// TIA Portal V16 export
// export: Created 2021-11-12T13:32:19.7443046Z, ExportSetting WithDefaults, DisplayName Totally Integrated Automation Portal, DisplayVersion V16 Update 3, DisplayName TIA Portal Version Control Interface, DisplayVersion V16 Update 2, DisplayName TIA Portal Openness, DisplayVersion V16 Update 3, DisplayName SINAMICS Startdrive Advanced, DisplayVersion V16 Update 5, DisplayName SINAMICS Startdrive G130, G150, S120, S150, SINAMICS MV, S210, DisplayVersion V16 Update 5, DisplayName SINAMICS Startdrive G110M, G120, G120C, G120D, G120P, G115D, DisplayVersion V16 Update 5, DisplayName STEP 7 Professional, DisplayVersion V16 Update 3, DisplayName STEP 7 Safety, DisplayVersion V16, DisplayName WinCC UA Professional, DisplayVersion V16 Update 3
FUNCTION_BLOCK "Station1R5"   // FB33, LAD
{ S7_Optimized_Access := 'TRUE' }
VERSION : 0.1
// stored: AutoNumber true, IsIECCheckEnabled false, IsRetainMemResEnabled false, MemoryReserve 100, SetENOAutomatically false, UDAEnableTagReadback false
   VAR
      SF_RO01_Timeout : "STD_DI_Mon";   // Move timeout
      "SF_CL01-BG01_Alarm" { S7_SetPoint := 'True'} : "STD_DI_Mon";
      "SF_CL01-BG02_Alarm" { S7_SetPoint := 'True'} : "STD_DI_Mon";
      SF_RC01 : "STD_DriveRobotABB";
      SF_RO01 : "STD_RobotABB";
      SF_RobotGripper : "STD_RobotGripper";
      SS_Edge { ExternalAccessible := 'False'; ExternalVisible := 'False'; ExternalWritable := 'False'} : Array[0..100] of Bool;
   END_VAR
   VAR RETAIN
      SDIPartID : DInt;
      SI_PartType { S7_SetPoint := 'True'} : Int;
   END_VAR
   VAR
      SI_150RowNr : Int;   // Row number in map of station 150
      SI_150LineNr : Int;   // Line number in map of station 150
      SI_170RowNr : Int;   // Row number in map of station 170
      SI_170LineNr : Int;   // Line number in map of station 170
      SI_BSN1BeltExt : Int;   // BSN1 belt extension
      SB1PosFound150 : Bool;   // Take position in map of station 150 found
      SB1PosFound170 : Bool;   // Take position in map of station 170 found
      SB1ReqToChangeTool : Bool;   // Request from zone command to change tools
      SB1ChangeToolDone : Bool;   // Changing tool process done
      SB1CycleAutostop : Bool;   // Cycle autostop command
      SB1ServicePosReq { ExternalAccessible := 'False'; ExternalVisible := 'False'; ExternalWritable := 'False'} : Bool;   // Request to go to/from service position
      SB1RobotInitialized : Bool;   // Robot is initialized
   END_VAR
   VAR_TEMP
      TS_RC01 : "UDT_DriveRobotABBControl";   // Robot controller RC01 control
      TS_RO01 : "UDT_RobotABBControl";   // Robot RO01 control
      TI_BSNJobNr : UInt;
      TI_RowNr : Int;   // Transfer mat card according to row number
      TI_LineNr : Int;   // Transfer mat card according to line number
      TB1PwrOK : Bool;   // Power for this station is OK
      TB1HomePosReq : Bool;   // Request to go to home position
      TB1CtrlRun : Bool;   // Robot controller is running in automat
      TB1GripperFree : Bool;   // Gripper free - info from robot and data tracking
      TB1Take150 : Bool;   // Take parts from 150
      TB1Take170 : Bool;   // Take parts from 170
      TB1PutBSN : Bool;   // Put parts BSN
      TB1ChangeToolUpDown : Bool;   // Change tool from CL01 to CL02
      TB1ChangeToolDownUp : Bool;   // Change tool from CL02 to CL01
      TB1FreePosBSN : Bool;   // Free position in furnace was found
      TB1JobNr150 : Bool;
      TB1JobNr170 : Bool;
   END_VAR
   VAR CONSTANT
      CI_JobHome : UInt := 1;
      CI_JobService : UInt := 2;
      CI_ChangeToolUpDown : UInt := 11;
      CI_ChangeToolDownUp : UInt := 12;
      CI_JobTake150Pos1 : UInt := 101;
      CI_JobTake150Pos2 : UInt := 102;
      CI_JobTake150Pos3 : UInt := 103;
      CI_JobTake150Pos4 : UInt := 104;
      CI_JobTake150Pos5 : UInt := 105;
      CI_JobTake150Pos6 : UInt := 106;
      CI_JobTake150Pos7 : UInt := 107;
      CI_JobTake150Pos8 : UInt := 108;
      CI_JobTake150Pos9 : UInt := 109;
      CI_JobTake150Pos10 : UInt := 110;
      CI_JobTake150Pos11 : UInt := 111;
      CI_JobTake150Pos12 : UInt := 112;
      CI_JobTake170Pos1 : UInt := 201;
      CI_JobTake170Pos2 : UInt := 202;
      CI_JobTake170Pos3 : UInt := 203;
      CI_JobTake170Pos4 : UInt := 204;
      CI_JobTake170Pos5 : UInt := 205;
      CI_JobTake170Pos6 : UInt := 206;
      CI_JobTake170Pos7 : UInt := 207;
      CI_JobTake170Pos8 : UInt := 208;
      CI_JobTake170Pos9 : UInt := 209;
      CI_JobTake170Pos10 : UInt := 210;
      CI_JobTake170Pos11 : UInt := 211;
      CI_JobTake170Pos12 : UInt := 212;
      CI_JobPutR12L12 : UInt := 301;
      CI_JobPutR12L23 : UInt := 302;
      CI_JobPutR12L34 : UInt := 303;
      CI_JobPutR12L45 : UInt := 304;
      CI_JobPutR23L12 : UInt := 305;
      CI_JobPutR23L23 : UInt := 306;
      CI_JobPutR23L34 : UInt := 307;
      CI_JobPutR23L45 : UInt := 308;
      CI_JobPutR34L12 : UInt := 309;
      CI_JobPutR34L23 : UInt := 310;
      CI_JobPutR34L34 : UInt := 311;
      CI_JobPutR34L45 : UInt := 312;
      CI_JobPutPosX : UInt := 313;
   END_VAR
   VAR_TEMP   // added for the SCL form of the ladder/FBD networks
      _w1 : Bool;
      _w2 : Bool;
      _w3 : Bool;
      _w4 : Bool;
      _w5 : Bool;
      _w6 : Bool;
      _w7 : Bool;
      _w8 : Bool;
      _w9 : Bool;
      _w10 : Bool;
      _w11 : Bool;
      _w12 : Bool;
      _w13 : Bool;
      _w14 : Bool;
   END_VAR
BEGIN

REGION Network 1: Clear temporary variables
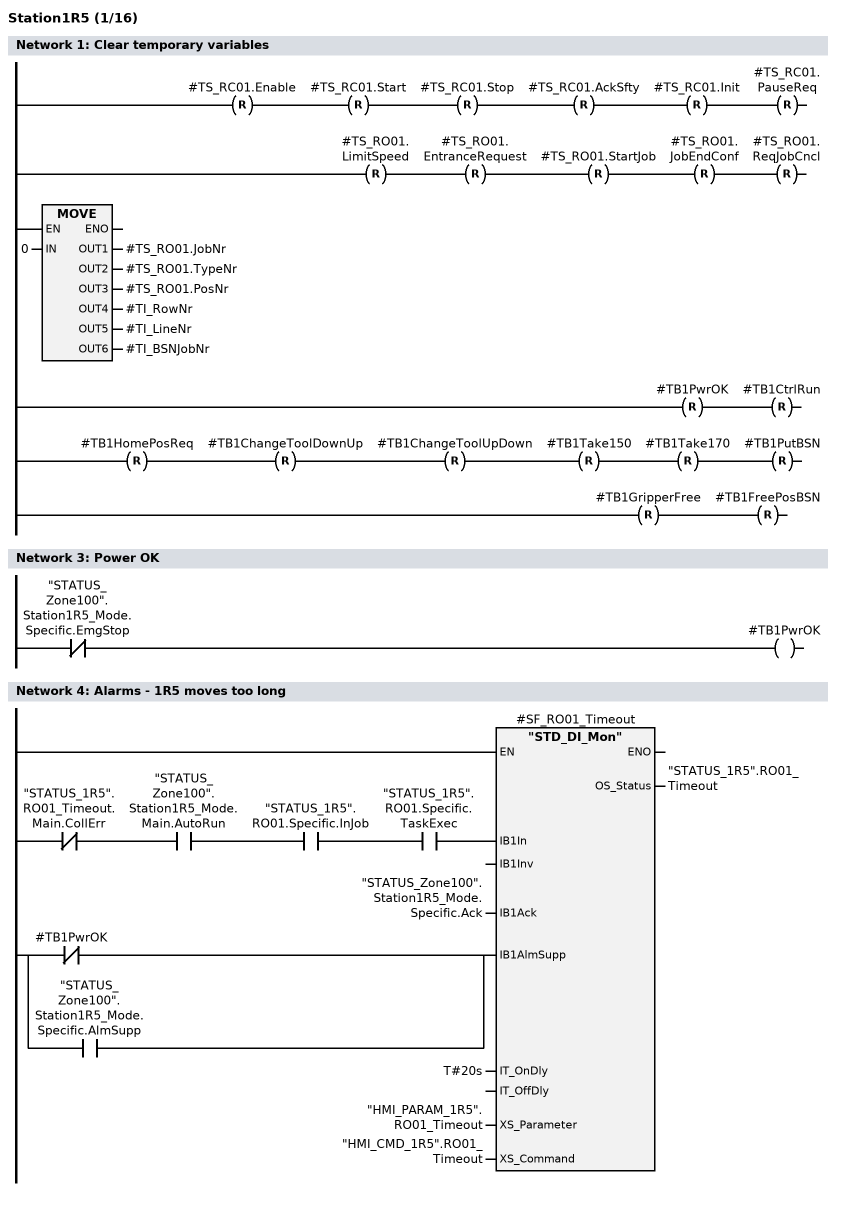
   RUNG wire#powerrail
      R_Coil( #TS_RC01.Enable )
      R_Coil( #TS_RC01.Start )
      R_Coil( #TS_RC01.Stop )
      R_Coil( #TS_RC01.AckSfty )
      R_Coil( #TS_RC01.Init )
      R_Coil( #TS_RC01.PauseReq )
   END_RUNG
   RUNG wire#powerrail
      R_Coil( #TS_RO01.LimitSpeed )
      R_Coil( #TS_RO01.EntranceRequest )
      R_Coil( #TS_RO01.StartJob )
      R_Coil( #TS_RO01.JobEndConf )
      R_Coil( #TS_RO01.ReqJobCncl )
   END_RUNG
   RUNG wire#powerrail
      Move(in := 0, out1 => #TS_RO01.JobNr, out2 => #TS_RO01.TypeNr, out3 => #TS_RO01.PosNr, out4 => #TI_RowNr, out5 => #TI_LineNr, out6 => #TI_BSNJobNr)
   END_RUNG
   RUNG wire#powerrail
      R_Coil( #TB1PwrOK )
      R_Coil( #TB1CtrlRun )
   END_RUNG
   RUNG wire#powerrail
      R_Coil( #TB1HomePosReq )
      R_Coil( #TB1ChangeToolDownUp )
      R_Coil( #TB1ChangeToolUpDown )
      R_Coil( #TB1Take150 )
      R_Coil( #TB1Take170 )
      R_Coil( #TB1PutBSN )
   END_RUNG
   RUNG wire#powerrail
      R_Coil( #TB1GripperFree )
      R_Coil( #TB1FreePosBSN )
   END_RUNG
   // the same network as SCL:
   #TS_RC01.Enable := FALSE;
   #TS_RC01.Start := FALSE;
   #TS_RC01.Stop := FALSE;
   #TS_RC01.AckSfty := FALSE;
   #TS_RC01.Init := FALSE;
   #TS_RC01.PauseReq := FALSE;
   #TS_RO01.LimitSpeed := FALSE;
   #TS_RO01.EntranceRequest := FALSE;
   #TS_RO01.StartJob := FALSE;
   #TS_RO01.JobEndConf := FALSE;
   #TS_RO01.ReqJobCncl := FALSE;
   #TS_RO01.JobNr := 0;
   #TS_RO01.TypeNr := 0;
   #TS_RO01.PosNr := 0;
   #TI_RowNr := 0;
   #TI_LineNr := 0;
   #TI_BSNJobNr := 0;
   #TB1PwrOK := FALSE;
   #TB1CtrlRun := FALSE;
   #TB1HomePosReq := FALSE;
   #TB1ChangeToolDownUp := FALSE;
   #TB1ChangeToolUpDown := FALSE;
   #TB1Take150 := FALSE;
   #TB1Take170 := FALSE;
   #TB1PutBSN := FALSE;
   #TB1GripperFree := FALSE;
   #TB1FreePosBSN := FALSE;
END_REGION

REGION Network 2: *************** Alarms ***************
END_REGION

REGION Network 3: Power OK
   RUNG wire#powerrail
      I_Contact( "STATUS_Zone100".Station1R5_Mode.Specific.EmgStop )
      Coil( #TB1PwrOK )
   END_RUNG
   // the same network as SCL:
   #TB1PwrOK := NOT "STATUS_Zone100".Station1R5_Mode.Specific.EmgStop;
END_REGION

REGION Network 4: Alarms - 1R5 moves too long
   RUNG wire#powerrail
      #SF_RO01_Timeout(IB1In := wire#w1, IB1AlmSupp := wire#w2, IB1Inv :=, IB1Ack := "STATUS_Zone100".Station1R5_Mode.Specific.Ack, IT_OnDly := T#20s, IT_OffDly :=, XS_Parameter := "HMI_PARAM_1R5".RO01_Timeout, XS_Command := "HMI_CMD_1R5".RO01_Timeout, OS_Status => "STATUS_1R5".RO01_Timeout)
   END_RUNG
   RUNG wire#powerrail
      I_Contact( "STATUS_1R5".RO01_Timeout.Main.CollErr )
      Contact( "STATUS_Zone100".Station1R5_Mode.Main.AutoRun )
      Contact( "STATUS_1R5".RO01.Specific.InJob )
      Contact( "STATUS_1R5".RO01.Specific.TaskExec )
   END_RUNG wire#w1
   RUNG wire#powerrail
      I_Contact( #TB1PwrOK )
   END_RUNG wire#w2
   RUNG wire#powerrail
      Contact( "STATUS_Zone100".Station1R5_Mode.Specific.AlmSupp )
   END_RUNG wire#w2
   // the same network as SCL:
   #SF_RO01_Timeout(IB1In := NOT "STATUS_1R5".RO01_Timeout.Main.CollErr AND "STATUS_Zone100".Station1R5_Mode.Main.AutoRun AND "STATUS_1R5".RO01.Specific.InJob AND "STATUS_1R5".RO01.Specific.TaskExec,   // "STD_DI_Mon"
                    IB1Ack := "STATUS_Zone100".Station1R5_Mode.Specific.Ack,
                    IB1AlmSupp := NOT #TB1PwrOK OR "STATUS_Zone100".Station1R5_Mode.Specific.AlmSupp,
                    IT_OnDly := T#20s,
                    XS_Parameter := "HMI_PARAM_1R5".RO01_Timeout,
                    XS_Command := "HMI_CMD_1R5".RO01_Timeout,
                    OS_Status => "STATUS_1R5".RO01_Timeout);
END_REGION

REGION Network 5: Sensor alarms - CL01
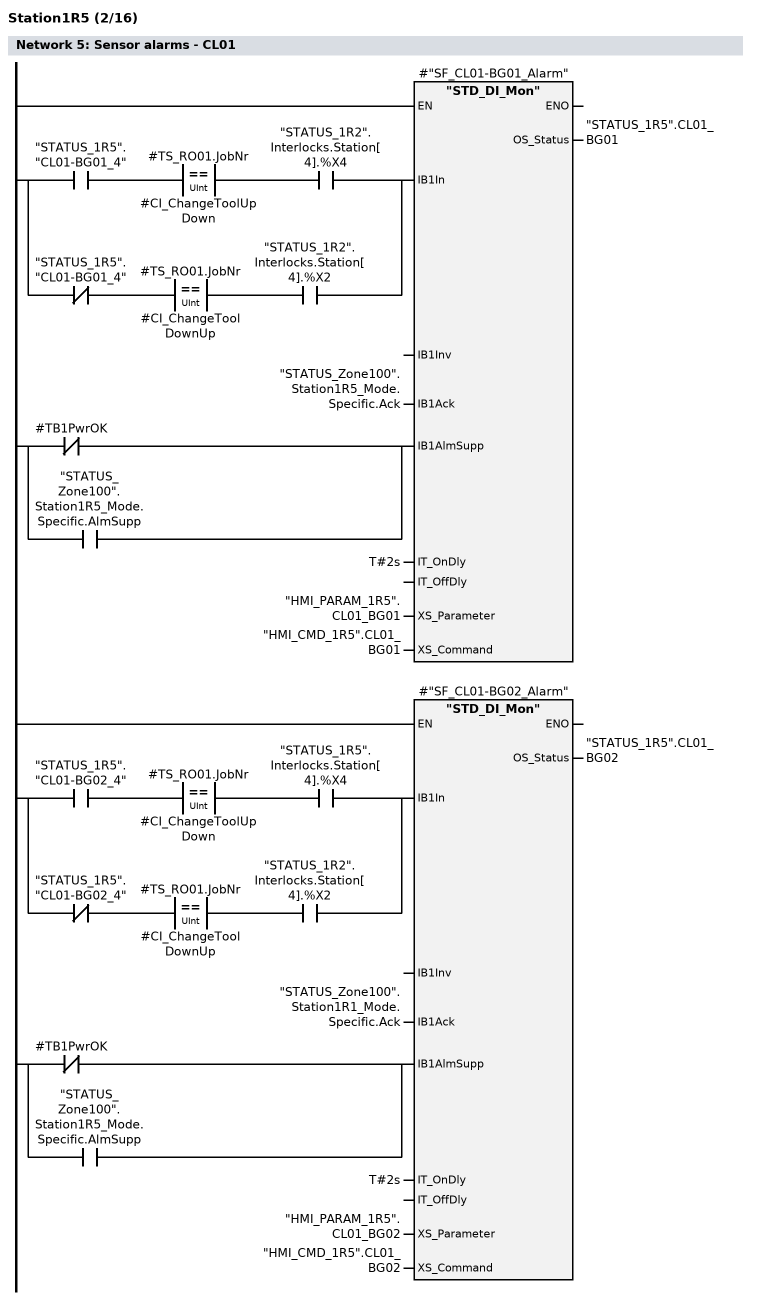
   RUNG wire#powerrail
      #"SF_CL01-BG01_Alarm"(IB1In := wire#w1, IB1AlmSupp := wire#w2, IB1Inv :=, IB1Ack := "STATUS_Zone100".Station1R5_Mode.Specific.Ack, IT_OnDly := T#2s, IT_OffDly :=, XS_Parameter := "HMI_PARAM_1R5".CL01_BG01, XS_Command := "HMI_CMD_1R5".CL01_BG01, OS_Status => "STATUS_1R5".CL01_BG01)
   END_RUNG
   RUNG wire#powerrail
      Contact( "STATUS_1R5"."CL01-BG01_4" )
      { S7_Templates := "SrcType := UInt" } EQ_Contact(in1 := #TS_RO01.JobNr, in2 := #CI_ChangeToolUpDown)
      Contact( "STATUS_1R2".Interlocks.Station[4].%X4 )
   END_RUNG wire#w1
   RUNG wire#powerrail
      I_Contact( "STATUS_1R5"."CL01-BG01_4" )
      { S7_Templates := "SrcType := UInt" } EQ_Contact(in1 := #TS_RO01.JobNr, in2 := #CI_ChangeToolDownUp)
      Contact( "STATUS_1R2".Interlocks.Station[4].%X2 )
   END_RUNG wire#w1
   RUNG wire#powerrail
      I_Contact( #TB1PwrOK )
   END_RUNG wire#w2
   RUNG wire#powerrail
      Contact( "STATUS_Zone100".Station1R5_Mode.Specific.AlmSupp )
   END_RUNG wire#w2
   RUNG wire#powerrail
      #"SF_CL01-BG02_Alarm"(IB1In := wire#w3, IB1AlmSupp := wire#w4, IB1Inv :=, IB1Ack := "STATUS_Zone100".Station1R1_Mode.Specific.Ack, IT_OnDly := T#2s, IT_OffDly :=, XS_Parameter := "HMI_PARAM_1R5".CL01_BG02, XS_Command := "HMI_CMD_1R5".CL01_BG02, OS_Status => "STATUS_1R5".CL01_BG02)
   END_RUNG
   RUNG wire#powerrail
      Contact( "STATUS_1R5"."CL01-BG02_4" )
      { S7_Templates := "SrcType := UInt" } EQ_Contact(in1 := #TS_RO01.JobNr, in2 := #CI_ChangeToolUpDown)
      Contact( "STATUS_1R5".Interlocks.Station[4].%X4 )
   END_RUNG wire#w3
   RUNG wire#powerrail
      I_Contact( "STATUS_1R5"."CL01-BG02_4" )
      { S7_Templates := "SrcType := UInt" } EQ_Contact(in1 := #TS_RO01.JobNr, in2 := #CI_ChangeToolDownUp)
      Contact( "STATUS_1R2".Interlocks.Station[4].%X2 )
   END_RUNG wire#w3
   RUNG wire#powerrail
      I_Contact( #TB1PwrOK )
   END_RUNG wire#w4
   RUNG wire#powerrail
      Contact( "STATUS_Zone100".Station1R5_Mode.Specific.AlmSupp )
   END_RUNG wire#w4
   // the same network as SCL:
   #"SF_CL01-BG01_Alarm"(IB1In := ("STATUS_1R5"."CL01-BG01_4" AND (#TS_RO01.JobNr = #CI_ChangeToolUpDown) AND "STATUS_1R2".Interlocks.Station[4].%X4) OR (NOT "STATUS_1R5"."CL01-BG01_4" AND (#TS_RO01.JobNr = #CI_ChangeToolDownUp) AND "STATUS_1R2".Interlocks.Station[4].%X2),   // "STD_DI_Mon"
                         IB1Ack := "STATUS_Zone100".Station1R5_Mode.Specific.Ack,
                         IB1AlmSupp := NOT #TB1PwrOK OR "STATUS_Zone100".Station1R5_Mode.Specific.AlmSupp,
                         IT_OnDly := T#2s,
                         XS_Parameter := "HMI_PARAM_1R5".CL01_BG01,
                         XS_Command := "HMI_CMD_1R5".CL01_BG01,
                         OS_Status => "STATUS_1R5".CL01_BG01);
   #"SF_CL01-BG02_Alarm"(IB1In := ("STATUS_1R5"."CL01-BG02_4" AND (#TS_RO01.JobNr = #CI_ChangeToolUpDown) AND "STATUS_1R5".Interlocks.Station[4].%X4) OR (NOT "STATUS_1R5"."CL01-BG02_4" AND (#TS_RO01.JobNr = #CI_ChangeToolDownUp) AND "STATUS_1R2".Interlocks.Station[4].%X2),   // "STD_DI_Mon"
                         IB1Ack := "STATUS_Zone100".Station1R1_Mode.Specific.Ack,
                         IB1AlmSupp := NOT #TB1PwrOK OR "STATUS_Zone100".Station1R5_Mode.Specific.AlmSupp,
                         IT_OnDly := T#2s,
                         XS_Parameter := "HMI_PARAM_1R5".CL01_BG02,
                         XS_Command := "HMI_CMD_1R5".CL01_BG02,
                         OS_Status => "STATUS_1R5".CL01_BG02);
END_REGION

REGION Network 6: *************** Controller RC01 ***************
END_REGION

REGION Network 7: Controller RC01 - control
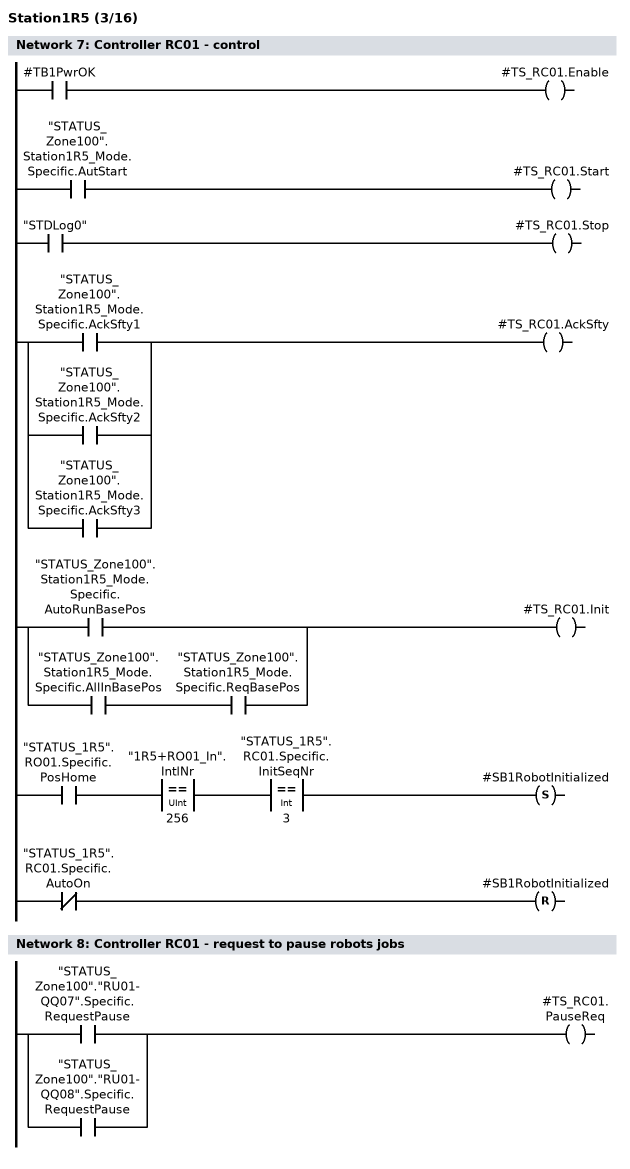
   RUNG wire#powerrail
      Contact( #TB1PwrOK )
      Coil( #TS_RC01.Enable )
   END_RUNG
   RUNG wire#powerrail
      Contact( "STATUS_Zone100".Station1R5_Mode.Specific.AutStart )
      Coil( #TS_RC01.Start )
   END_RUNG
   RUNG wire#powerrail
      Contact( "STDLog0" )
      Coil( #TS_RC01.Stop )
   END_RUNG
   RUNG wire#powerrail
      Contact( "STATUS_Zone100".Station1R5_Mode.Specific.AckSfty1 )
      wire#w1
      Coil( #TS_RC01.AckSfty )
   END_RUNG
   RUNG wire#powerrail
      Contact( "STATUS_Zone100".Station1R5_Mode.Specific.AckSfty2 )
   END_RUNG wire#w1
   RUNG wire#powerrail
      Contact( "STATUS_Zone100".Station1R5_Mode.Specific.AckSfty3 )
   END_RUNG wire#w1
   RUNG wire#powerrail
      Contact( "STATUS_Zone100".Station1R5_Mode.Specific.AutoRunBasePos )
      wire#w2
      Coil( #TS_RC01.Init )
   END_RUNG
   RUNG wire#powerrail
      Contact( "STATUS_Zone100".Station1R5_Mode.Specific.AllInBasePos )
      Contact( "STATUS_Zone100".Station1R5_Mode.Specific.ReqBasePos )
   END_RUNG wire#w2
   RUNG wire#powerrail
      Contact( "STATUS_1R5".RO01.Specific.PosHome )
      { S7_Templates := "SrcType := UInt" } EQ_Contact(in1 := "1R5+RO01_In".IntlNr, in2 := 256)
      { S7_Templates := "SrcType := Int" } EQ_Contact(in1 := "STATUS_1R5".RC01.Specific.InitSeqNr, in2 := 3)
      S_Coil( #SB1RobotInitialized )
   END_RUNG
   RUNG wire#powerrail
      I_Contact( "STATUS_1R5".RC01.Specific.AutoOn )
      R_Coil( #SB1RobotInitialized )
   END_RUNG
   // the same network as SCL:
   #TS_RC01.Enable := #TB1PwrOK;
   #TS_RC01.Start := "STATUS_Zone100".Station1R5_Mode.Specific.AutStart;
   #TS_RC01.Stop := "STDLog0";
   #TS_RC01.AckSfty := "STATUS_Zone100".Station1R5_Mode.Specific.AckSfty1 OR "STATUS_Zone100".Station1R5_Mode.Specific.AckSfty2 OR "STATUS_Zone100".Station1R5_Mode.Specific.AckSfty3;
   #TS_RC01.Init := "STATUS_Zone100".Station1R5_Mode.Specific.AutoRunBasePos OR ("STATUS_Zone100".Station1R5_Mode.Specific.AllInBasePos AND "STATUS_Zone100".Station1R5_Mode.Specific.ReqBasePos);
   IF "STATUS_1R5".RO01.Specific.PosHome AND ("1R5+RO01_In".IntlNr = 256) AND ("STATUS_1R5".RC01.Specific.InitSeqNr = 3) THEN
       #SB1RobotInitialized := TRUE;
   END_IF;
   IF NOT "STATUS_1R5".RC01.Specific.AutoOn THEN #SB1RobotInitialized := FALSE; END_IF;
END_REGION

REGION Network 8: Controller RC01 - request to pause robots jobs
   RUNG wire#powerrail
      Contact( "STATUS_Zone100"."RU01-QQ07".Specific.RequestPause )
      wire#w1
      Coil( #TS_RC01.PauseReq )
   END_RUNG
   RUNG wire#powerrail
      Contact( "STATUS_Zone100"."RU01-QQ08".Specific.RequestPause )
   END_RUNG wire#w1
   // the same network as SCL:
   #TS_RC01.PauseReq := "STATUS_Zone100"."RU01-QQ07".Specific.RequestPause OR "STATUS_Zone100"."RU01-QQ08".Specific.RequestPause;
END_REGION

REGION Network 9: Controller RC01 - main control
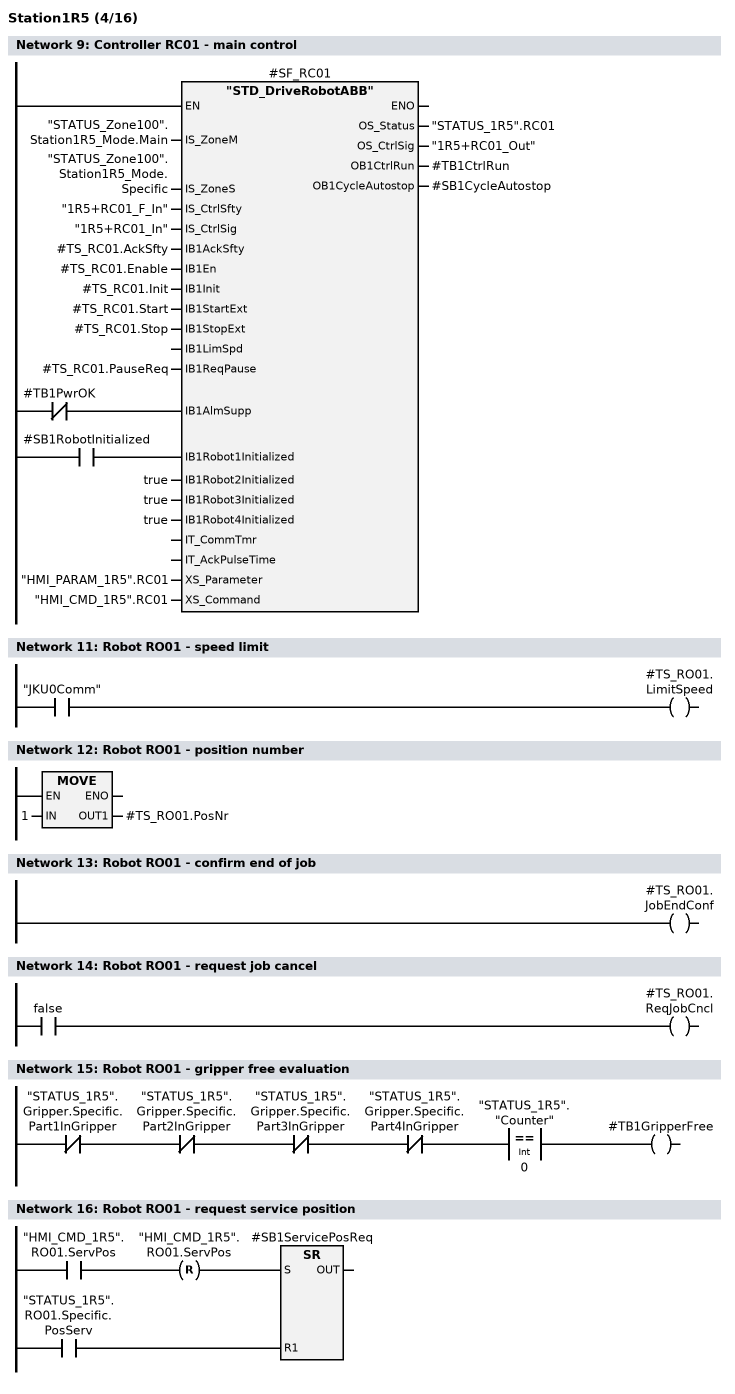
   RUNG wire#powerrail
      #SF_RC01(IB1AlmSupp := wire#w1, IB1Robot1Initialized := wire#w2, IS_ZoneM := "STATUS_Zone100".Station1R5_Mode.Main, IS_ZoneS := "STATUS_Zone100".Station1R5_Mode.Specific, IS_CtrlSfty := "1R5+RC01_F_In", IS_CtrlSig := "1R5+RC01_In", IB1AckSfty := #TS_RC01.AckSfty, IB1En := #TS_RC01.Enable, IB1Init := #TS_RC01.Init, IB1StartExt := #TS_RC01.Start, IB1StopExt := #TS_RC01.Stop, IB1LimSpd :=, IB1ReqPause := #TS_RC01.PauseReq, IB1Robot2Initialized := true, IB1Robot3Initialized := true, IB1Robot4Initialized := true, IT_CommTmr :=, IT_AckPulseTime :=, XS_Parameter := "HMI_PARAM_1R5".RC01, XS_Command := "HMI_CMD_1R5".RC01, OS_Status => "STATUS_1R5".RC01, OS_CtrlSig => "1R5+RC01_Out", OB1CtrlRun => #TB1CtrlRun, OB1CycleAutostop => #SB1CycleAutostop)
   END_RUNG
   RUNG wire#powerrail
      I_Contact( #TB1PwrOK )
   END_RUNG wire#w1
   RUNG wire#powerrail
      Contact( #SB1RobotInitialized )
   END_RUNG wire#w2
   // the same network as SCL:
   #SF_RC01(IS_ZoneM := "STATUS_Zone100".Station1R5_Mode.Main,   // "STD_DriveRobotABB"
            IS_ZoneS := "STATUS_Zone100".Station1R5_Mode.Specific,
            IS_CtrlSfty := "1R5+RC01_F_In",
            IS_CtrlSig := "1R5+RC01_In",
            IB1AckSfty := #TS_RC01.AckSfty,
            IB1En := #TS_RC01.Enable,
            IB1Init := #TS_RC01.Init,
            IB1StartExt := #TS_RC01.Start,
            IB1StopExt := #TS_RC01.Stop,
            IB1ReqPause := #TS_RC01.PauseReq,
            IB1AlmSupp := NOT #TB1PwrOK,
            IB1Robot1Initialized := #SB1RobotInitialized,
            IB1Robot2Initialized := true,
            IB1Robot3Initialized := true,
            IB1Robot4Initialized := true,
            XS_Parameter := "HMI_PARAM_1R5".RC01,
            XS_Command := "HMI_CMD_1R5".RC01,
            OS_Status => "STATUS_1R5".RC01,
            OS_CtrlSig => "1R5+RC01_Out",
            OB1CtrlRun => #TB1CtrlRun,
            OB1CycleAutostop => #SB1CycleAutostop);
END_REGION

REGION Network 10: *************** Robot RO01 ***************
END_REGION

REGION Network 11: Robot RO01 - speed limit
   RUNG wire#powerrail
      Contact( "JKU0Comm" )
      Coil( #TS_RO01.LimitSpeed )
   END_RUNG
   // the same network as SCL:
   #TS_RO01.LimitSpeed := "JKU0Comm";
END_REGION

REGION Network 12: Robot RO01 - position number
   RUNG wire#powerrail
      Move(in := 1, out1 => #TS_RO01.PosNr)
   END_RUNG
   // the same network as SCL:
   #TS_RO01.PosNr := 1;
END_REGION

REGION Network 13: Robot RO01 - confirm end of job
   RUNG wire#powerrail
      Coil( #TS_RO01.JobEndConf )
   END_RUNG
   // the same network as SCL:
   #TS_RO01.JobEndConf := TRUE;
END_REGION

REGION Network 14: Robot RO01 - request job cancel
   RUNG wire#powerrail
      Contact( false )
      Coil( #TS_RO01.ReqJobCncl )
   END_RUNG
   // the same network as SCL:
   #TS_RO01.ReqJobCncl := false;
END_REGION

REGION Network 15: Robot RO01 - gripper free evaluation
   RUNG wire#powerrail
      I_Contact( "STATUS_1R5".Gripper.Specific.Part1InGripper )
      I_Contact( "STATUS_1R5".Gripper.Specific.Part2InGripper )
      I_Contact( "STATUS_1R5".Gripper.Specific.Part3InGripper )
      I_Contact( "STATUS_1R5".Gripper.Specific.Part4InGripper )
      { S7_Templates := "SrcType := Int" } EQ_Contact(in1 := "STATUS_1R5"."Counter", in2 := 0)
      Coil( #TB1GripperFree )
   END_RUNG
   // the same network as SCL:
   #TB1GripperFree := NOT "STATUS_1R5".Gripper.Specific.Part1InGripper AND NOT "STATUS_1R5".Gripper.Specific.Part2InGripper AND NOT "STATUS_1R5".Gripper.Specific.Part3InGripper AND NOT "STATUS_1R5".Gripper.Specific.Part4InGripper AND ("STATUS_1R5"."Counter" = 0);
END_REGION

REGION Network 16: Robot RO01 - request service position
   RUNG wire#powerrail
      Contact( "HMI_CMD_1R5".RO01.ServPos )
      R_Coil( "HMI_CMD_1R5".RO01.ServPos )
      S_SR(operand := #SB1ServicePosReq, r1 := wire#w1)
   END_RUNG
   RUNG wire#powerrail
      Contact( "STATUS_1R5".RO01.Specific.PosServ )
   END_RUNG wire#w1
   // the same network as SCL:
   #_w1 := "HMI_CMD_1R5".RO01.ServPos;
   IF #_w1 THEN
       "HMI_CMD_1R5".RO01.ServPos := FALSE;
       #SB1ServicePosReq := TRUE;   // SR flip-flop
   END_IF;
   IF "STATUS_1R5".RO01.Specific.PosServ THEN #SB1ServicePosReq := FALSE; END_IF;
END_REGION

REGION Network 17: Robot RO01 - request home position
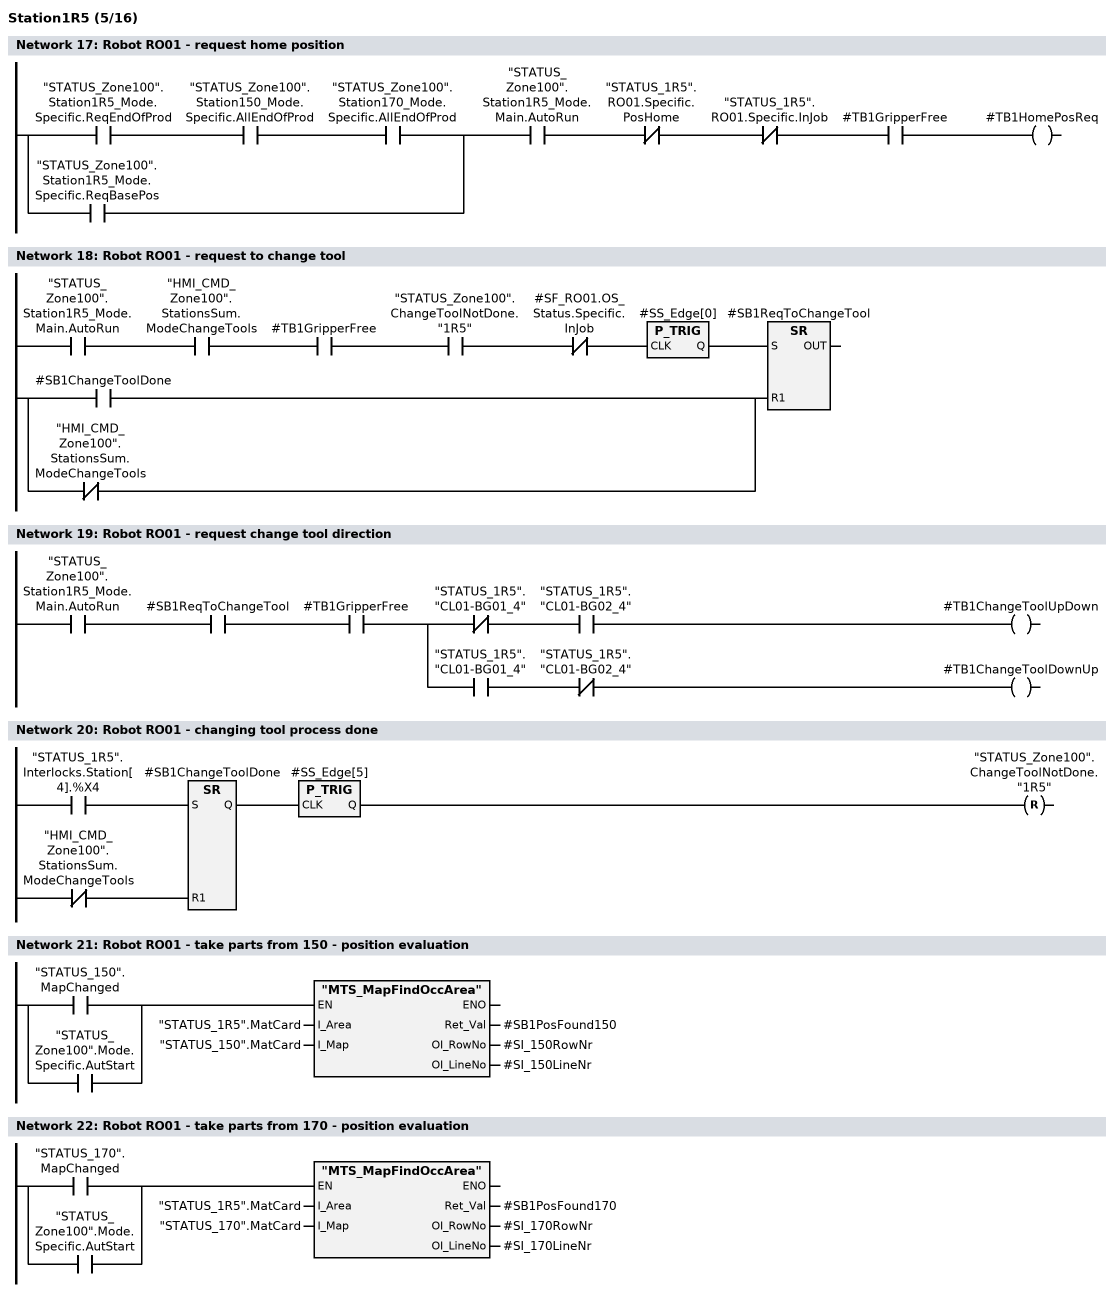
   RUNG wire#powerrail
      Contact( "STATUS_Zone100".Station1R5_Mode.Specific.ReqEndOfProd )
      Contact( "STATUS_Zone100".Station150_Mode.Specific.AllEndOfProd )
      Contact( "STATUS_Zone100".Station170_Mode.Specific.AllEndOfProd )
      wire#w1
      Contact( "STATUS_Zone100".Station1R5_Mode.Main.AutoRun )
      I_Contact( "STATUS_1R5".RO01.Specific.PosHome )
      I_Contact( "STATUS_1R5".RO01.Specific.InJob )
      Contact( #TB1GripperFree )
      Coil( #TB1HomePosReq )
   END_RUNG
   RUNG wire#powerrail
      Contact( "STATUS_Zone100".Station1R5_Mode.Specific.ReqBasePos )
   END_RUNG wire#w1
   // the same network as SCL:
   #TB1HomePosReq := (("STATUS_Zone100".Station1R5_Mode.Specific.ReqEndOfProd AND "STATUS_Zone100".Station150_Mode.Specific.AllEndOfProd AND "STATUS_Zone100".Station170_Mode.Specific.AllEndOfProd) OR "STATUS_Zone100".Station1R5_Mode.Specific.ReqBasePos) AND "STATUS_Zone100".Station1R5_Mode.Main.AutoRun AND NOT "STATUS_1R5".RO01.Specific.PosHome AND NOT "STATUS_1R5".RO01.Specific.InJob AND #TB1GripperFree;
END_REGION

REGION Network 18: Robot RO01 - request to change tool
   RUNG wire#powerrail
      Contact( "STATUS_Zone100".Station1R5_Mode.Main.AutoRun )
      Contact( "HMI_CMD_Zone100".StationsSum.ModeChangeTools )
      Contact( #TB1GripperFree )
      Contact( "STATUS_Zone100".ChangeToolNotDone."1R5" )
      I_Contact( #SF_RO01.OS_Status.Specific.InJob )
      P_Trig( #SS_Edge[0] )
      S_SR(operand := #SB1ReqToChangeTool, r1 := wire#w1)
   END_RUNG
   RUNG wire#powerrail
      Contact( #SB1ChangeToolDone )
   END_RUNG wire#w1
   RUNG wire#powerrail
      I_Contact( "HMI_CMD_Zone100".StationsSum.ModeChangeTools )
   END_RUNG wire#w1
   // the same network as SCL:
   #_w1 := "STATUS_Zone100".Station1R5_Mode.Main.AutoRun AND "HMI_CMD_Zone100".StationsSum.ModeChangeTools AND #TB1GripperFree AND "STATUS_Zone100".ChangeToolNotDone."1R5" AND NOT #SF_RO01.OS_Status.Specific.InJob;
   #_w2 := #_w1 AND NOT #SS_Edge[0];   // rising edge
   #SS_Edge[0] := #_w1;
   IF #_w2 THEN
       #SB1ReqToChangeTool := TRUE;   // SR flip-flop
   END_IF;
   IF #SB1ChangeToolDone OR NOT "HMI_CMD_Zone100".StationsSum.ModeChangeTools THEN
       #SB1ReqToChangeTool := FALSE;
   END_IF;
END_REGION

REGION Network 19: Robot RO01 - request change tool direction
   RUNG wire#powerrail
      Contact( "STATUS_Zone100".Station1R5_Mode.Main.AutoRun )
      Contact( #SB1ReqToChangeTool )
      Contact( #TB1GripperFree )
      wire#w1
      I_Contact( "STATUS_1R5"."CL01-BG01_4" )
      Contact( "STATUS_1R5"."CL01-BG02_4" )
      Coil( #TB1ChangeToolUpDown )
   END_RUNG
   RUNG wire#w1
      Contact( "STATUS_1R5"."CL01-BG01_4" )
      I_Contact( "STATUS_1R5"."CL01-BG02_4" )
      Coil( #TB1ChangeToolDownUp )
   END_RUNG
   // the same network as SCL:
   #_w1 := "STATUS_Zone100".Station1R5_Mode.Main.AutoRun AND #SB1ReqToChangeTool AND #TB1GripperFree;
   #TB1ChangeToolUpDown := #_w1 AND NOT "STATUS_1R5"."CL01-BG01_4" AND "STATUS_1R5"."CL01-BG02_4";
   #TB1ChangeToolDownUp := #_w1 AND "STATUS_1R5"."CL01-BG01_4" AND NOT "STATUS_1R5"."CL01-BG02_4";
END_REGION

REGION Network 20: Robot RO01 - changing tool process done
   RUNG wire#powerrail
      Contact( "STATUS_1R5".Interlocks.Station[4].%X4 )
      S_SR(operand := #SB1ChangeToolDone, r1 := wire#w1)
      P_Trig( #SS_Edge[5] )
      R_Coil( "STATUS_Zone100".ChangeToolNotDone."1R5" )
   END_RUNG
   RUNG wire#powerrail
      I_Contact( "HMI_CMD_Zone100".StationsSum.ModeChangeTools )
   END_RUNG wire#w1
   // the same network as SCL:
   IF "STATUS_1R5".Interlocks.Station[4].%X4 THEN
       #SB1ChangeToolDone := TRUE;   // SR flip-flop
   END_IF;
   IF NOT "HMI_CMD_Zone100".StationsSum.ModeChangeTools THEN #SB1ChangeToolDone := FALSE; END_IF;
   #_w1 := #SB1ChangeToolDone AND NOT #SS_Edge[5];   // rising edge
   #SS_Edge[5] := #SB1ChangeToolDone;
   IF #_w1 THEN "STATUS_Zone100".ChangeToolNotDone."1R5" := FALSE; END_IF;
END_REGION

REGION Network 21: Robot RO01 - take parts from 150 - position evaluation
   RUNG wire#powerrail
      Contact( "STATUS_150".MapChanged )
      wire#w1
      "MTS_MapFindOccArea"(I_Area := "STATUS_1R5".MatCard, I_Map := "STATUS_150".MatCard, Ret_Val => #SB1PosFound150, OI_RowNo => #SI_150RowNr, OI_LineNo => #SI_150LineNr)
   END_RUNG
   RUNG wire#powerrail
      Contact( "STATUS_Zone100".Mode.Specific.AutStart )
   END_RUNG wire#w1
   // the same network as SCL:
   IF "STATUS_150".MapChanged OR "STATUS_Zone100".Mode.Specific.AutStart THEN
       #SB1PosFound150 := "MTS_MapFindOccArea"(I_Area := "STATUS_1R5".MatCard,
                               I_Map := "STATUS_150".MatCard,
                               OI_RowNo => #SI_150RowNr,
                               OI_LineNo => #SI_150LineNr);
   END_IF;
END_REGION

REGION Network 22: Robot RO01 - take parts from 170 - position evaluation
   RUNG wire#powerrail
      Contact( "STATUS_170".MapChanged )
      wire#w1
      "MTS_MapFindOccArea"(I_Area := "STATUS_1R5".MatCard, I_Map := "STATUS_170".MatCard, Ret_Val => #SB1PosFound170, OI_RowNo => #SI_170RowNr, OI_LineNo => #SI_170LineNr)
   END_RUNG
   RUNG wire#powerrail
      Contact( "STATUS_Zone100".Mode.Specific.AutStart )
   END_RUNG wire#w1
   // the same network as SCL:
   IF "STATUS_170".MapChanged OR "STATUS_Zone100".Mode.Specific.AutStart THEN
       #SB1PosFound170 := "MTS_MapFindOccArea"(I_Area := "STATUS_1R5".MatCard,
                               I_Map := "STATUS_170".MatCard,
                               OI_RowNo => #SI_170RowNr,
                               OI_LineNo => #SI_170LineNr);
   END_IF;
END_REGION

REGION Network 23: Robot RO01 - table 150/170 - take command
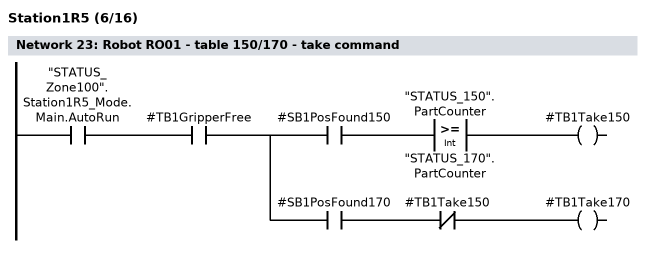
   RUNG wire#powerrail
      Contact( "STATUS_Zone100".Station1R5_Mode.Main.AutoRun )
      Contact( #TB1GripperFree )
      wire#w1
      Contact( #SB1PosFound150 )
      { S7_Templates := "SrcType := Int" } GE_Contact(in1 := "STATUS_150".PartCounter, in2 := "STATUS_170".PartCounter)
      Coil( #TB1Take150 )
   END_RUNG
   RUNG wire#w1
      Contact( #SB1PosFound170 )
      I_Contact( #TB1Take150 )
      Coil( #TB1Take170 )
   END_RUNG
   // the same network as SCL:
   #_w1 := "STATUS_Zone100".Station1R5_Mode.Main.AutoRun AND #TB1GripperFree;
   #TB1Take150 := #_w1 AND #SB1PosFound150 AND ("STATUS_150".PartCounter >= "STATUS_170".PartCounter);
   #TB1Take170 := #_w1 AND #SB1PosFound170 AND NOT #TB1Take150;
END_REGION

REGION Network 24: Robot RO01 - BSN1 position evaluation
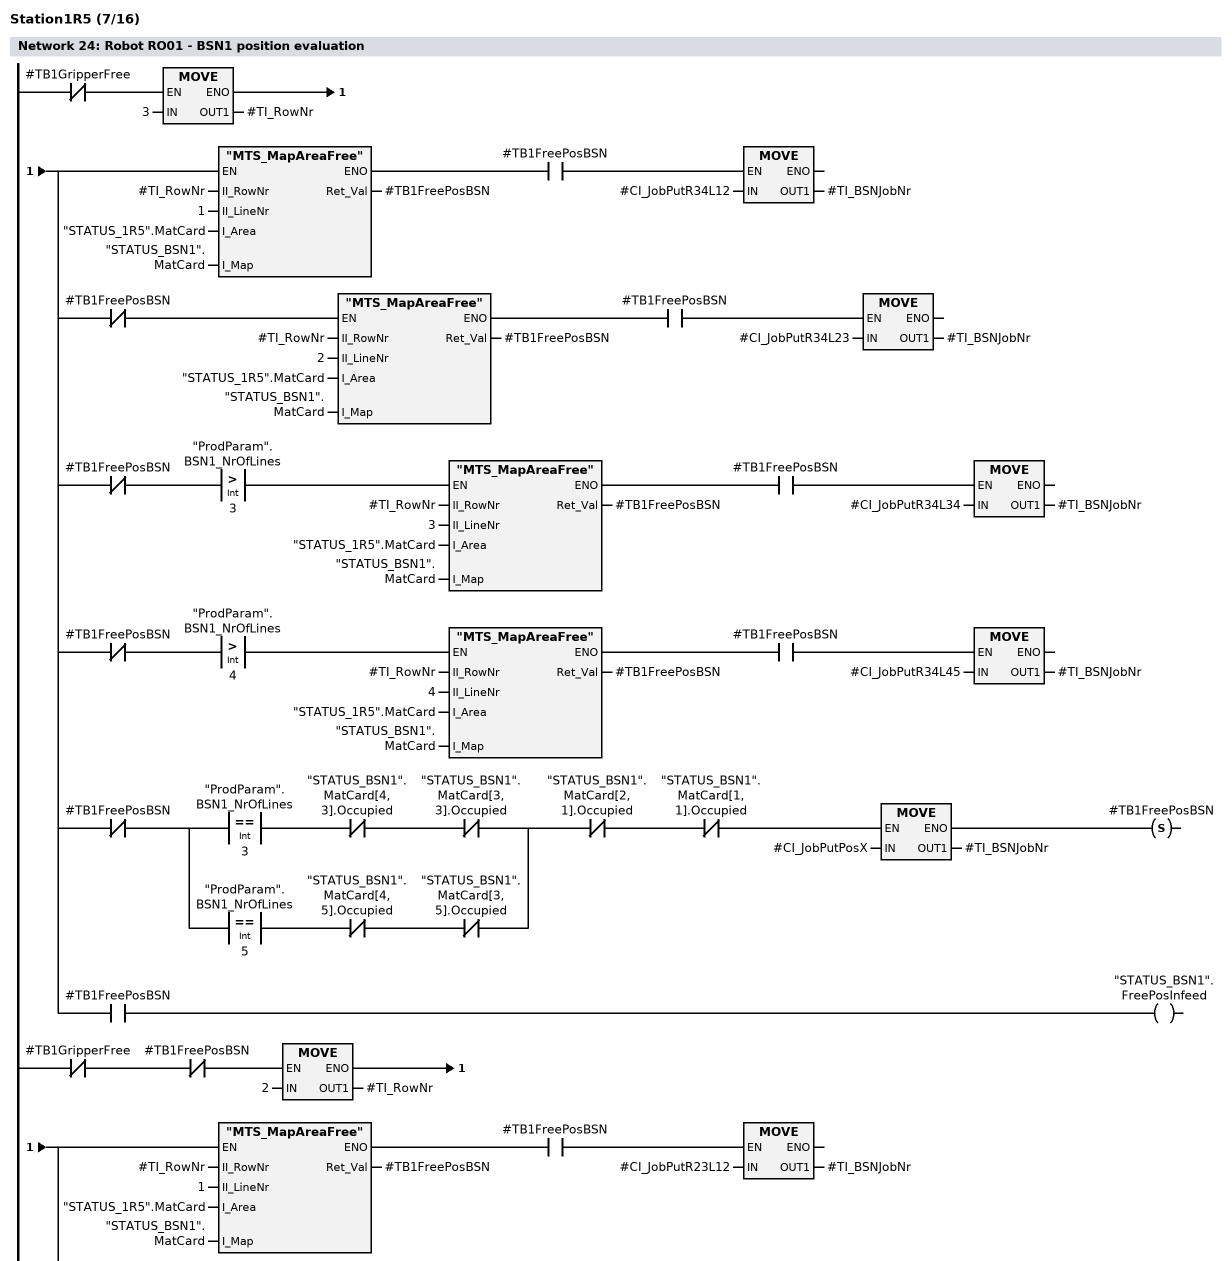
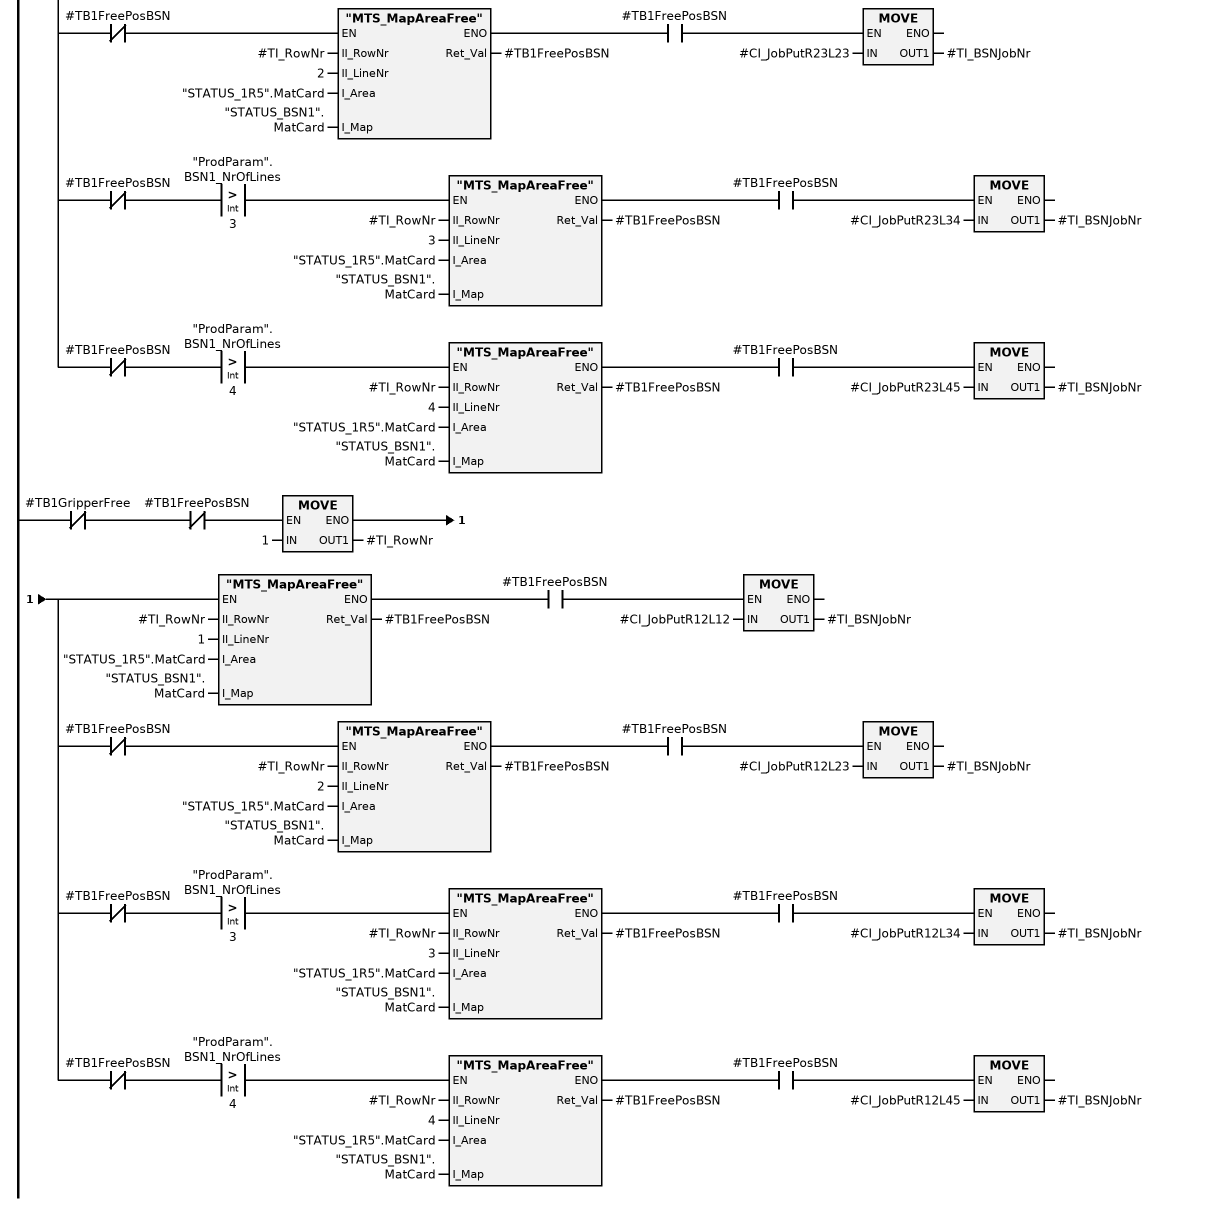
   RUNG wire#powerrail
      I_Contact( #TB1GripperFree )
      Move(in := 3, out1 => #TI_RowNr)
      wire#w1
      "MTS_MapAreaFree"(II_RowNr := #TI_RowNr, II_LineNr := 1, I_Area := "STATUS_1R5".MatCard, I_Map := "STATUS_BSN1".MatCard, Ret_Val => #TB1FreePosBSN)
      Contact( #TB1FreePosBSN )
      Move(in := #CI_JobPutR34L12, out1 => #TI_BSNJobNr)
   END_RUNG
   RUNG wire#w1
      I_Contact( #TB1FreePosBSN )
      "MTS_MapAreaFree"(II_RowNr := #TI_RowNr, II_LineNr := 2, I_Area := "STATUS_1R5".MatCard, I_Map := "STATUS_BSN1".MatCard, Ret_Val => #TB1FreePosBSN)
      Contact( #TB1FreePosBSN )
      Move(in := #CI_JobPutR34L23, out1 => #TI_BSNJobNr)
   END_RUNG
   RUNG wire#w1
      I_Contact( #TB1FreePosBSN )
      { S7_Templates := "SrcType := Int" } GT_Contact(in1 := "ProdParam".BSN1_NrOfLines, in2 := 3)
      "MTS_MapAreaFree"(II_RowNr := #TI_RowNr, II_LineNr := 3, I_Area := "STATUS_1R5".MatCard, I_Map := "STATUS_BSN1".MatCard, Ret_Val => #TB1FreePosBSN)
      Contact( #TB1FreePosBSN )
      Move(in := #CI_JobPutR34L34, out1 => #TI_BSNJobNr)
   END_RUNG
   RUNG wire#w1
      I_Contact( #TB1FreePosBSN )
      { S7_Templates := "SrcType := Int" } GT_Contact(in1 := "ProdParam".BSN1_NrOfLines, in2 := 4)
      "MTS_MapAreaFree"(II_RowNr := #TI_RowNr, II_LineNr := 4, I_Area := "STATUS_1R5".MatCard, I_Map := "STATUS_BSN1".MatCard, Ret_Val => #TB1FreePosBSN)
      Contact( #TB1FreePosBSN )
      Move(in := #CI_JobPutR34L45, out1 => #TI_BSNJobNr)
   END_RUNG
   RUNG wire#w1
      I_Contact( #TB1FreePosBSN )
      wire#w2
      { S7_Templates := "SrcType := Int" } EQ_Contact(in1 := "ProdParam".BSN1_NrOfLines, in2 := 3)
      I_Contact( "STATUS_BSN1".MatCard[4, 3].Occupied )
      I_Contact( "STATUS_BSN1".MatCard[3, 3].Occupied )
      wire#w3
      I_Contact( "STATUS_BSN1".MatCard[2, 1].Occupied )
      I_Contact( "STATUS_BSN1".MatCard[1, 1].Occupied )
      Move(in := #CI_JobPutPosX, out1 => #TI_BSNJobNr)
      S_Coil( #TB1FreePosBSN )
   END_RUNG
   RUNG wire#w2
      { S7_Templates := "SrcType := Int" } EQ_Contact(in1 := "ProdParam".BSN1_NrOfLines, in2 := 5)
      I_Contact( "STATUS_BSN1".MatCard[4, 5].Occupied )
      I_Contact( "STATUS_BSN1".MatCard[3, 5].Occupied )
   END_RUNG wire#w3
   RUNG wire#w1
      Contact( #TB1FreePosBSN )
      Coil( "STATUS_BSN1".FreePosInfeed )
   END_RUNG
   RUNG wire#powerrail
      I_Contact( #TB1GripperFree )
      I_Contact( #TB1FreePosBSN )
      Move(in := 2, out1 => #TI_RowNr)
      wire#w4
      "MTS_MapAreaFree"(II_RowNr := #TI_RowNr, II_LineNr := 1, I_Area := "STATUS_1R5".MatCard, I_Map := "STATUS_BSN1".MatCard, Ret_Val => #TB1FreePosBSN)
      Contact( #TB1FreePosBSN )
      Move(in := #CI_JobPutR23L12, out1 => #TI_BSNJobNr)
   END_RUNG
   RUNG wire#w4
      I_Contact( #TB1FreePosBSN )
      "MTS_MapAreaFree"(II_RowNr := #TI_RowNr, II_LineNr := 2, I_Area := "STATUS_1R5".MatCard, I_Map := "STATUS_BSN1".MatCard, Ret_Val => #TB1FreePosBSN)
      Contact( #TB1FreePosBSN )
      Move(in := #CI_JobPutR23L23, out1 => #TI_BSNJobNr)
   END_RUNG
   RUNG wire#w4
      I_Contact( #TB1FreePosBSN )
      { S7_Templates := "SrcType := Int" } GT_Contact(in1 := "ProdParam".BSN1_NrOfLines, in2 := 3)
      "MTS_MapAreaFree"(II_RowNr := #TI_RowNr, II_LineNr := 3, I_Area := "STATUS_1R5".MatCard, I_Map := "STATUS_BSN1".MatCard, Ret_Val => #TB1FreePosBSN)
      Contact( #TB1FreePosBSN )
      Move(in := #CI_JobPutR23L34, out1 => #TI_BSNJobNr)
   END_RUNG
   RUNG wire#w4
      I_Contact( #TB1FreePosBSN )
      { S7_Templates := "SrcType := Int" } GT_Contact(in1 := "ProdParam".BSN1_NrOfLines, in2 := 4)
      "MTS_MapAreaFree"(II_RowNr := #TI_RowNr, II_LineNr := 4, I_Area := "STATUS_1R5".MatCard, I_Map := "STATUS_BSN1".MatCard, Ret_Val => #TB1FreePosBSN)
      Contact( #TB1FreePosBSN )
      Move(in := #CI_JobPutR23L45, out1 => #TI_BSNJobNr)
   END_RUNG
   RUNG wire#powerrail
      I_Contact( #TB1GripperFree )
      I_Contact( #TB1FreePosBSN )
      Move(in := 1, out1 => #TI_RowNr)
      wire#w5
      "MTS_MapAreaFree"(II_RowNr := #TI_RowNr, II_LineNr := 1, I_Area := "STATUS_1R5".MatCard, I_Map := "STATUS_BSN1".MatCard, Ret_Val => #TB1FreePosBSN)
      Contact( #TB1FreePosBSN )
      Move(in := #CI_JobPutR12L12, out1 => #TI_BSNJobNr)
   END_RUNG
   RUNG wire#w5
      I_Contact( #TB1FreePosBSN )
      "MTS_MapAreaFree"(II_RowNr := #TI_RowNr, II_LineNr := 2, I_Area := "STATUS_1R5".MatCard, I_Map := "STATUS_BSN1".MatCard, Ret_Val => #TB1FreePosBSN)
      Contact( #TB1FreePosBSN )
      Move(in := #CI_JobPutR12L23, out1 => #TI_BSNJobNr)
   END_RUNG
   RUNG wire#w5
      I_Contact( #TB1FreePosBSN )
      { S7_Templates := "SrcType := Int" } GT_Contact(in1 := "ProdParam".BSN1_NrOfLines, in2 := 3)
      "MTS_MapAreaFree"(II_RowNr := #TI_RowNr, II_LineNr := 3, I_Area := "STATUS_1R5".MatCard, I_Map := "STATUS_BSN1".MatCard, Ret_Val => #TB1FreePosBSN)
      Contact( #TB1FreePosBSN )
      Move(in := #CI_JobPutR12L34, out1 => #TI_BSNJobNr)
   END_RUNG
   RUNG wire#w5
      I_Contact( #TB1FreePosBSN )
      { S7_Templates := "SrcType := Int" } GT_Contact(in1 := "ProdParam".BSN1_NrOfLines, in2 := 4)
      "MTS_MapAreaFree"(II_RowNr := #TI_RowNr, II_LineNr := 4, I_Area := "STATUS_1R5".MatCard, I_Map := "STATUS_BSN1".MatCard, Ret_Val => #TB1FreePosBSN)
      Contact( #TB1FreePosBSN )
      Move(in := #CI_JobPutR12L45, out1 => #TI_BSNJobNr)
   END_RUNG
   // the same network as SCL:
   IF NOT #TB1GripperFree THEN #TI_RowNr := 3; END_IF;
   #TB1FreePosBSN := "MTS_MapAreaFree"(EN := NOT #TB1GripperFree,
                           II_RowNr := #TI_RowNr,
                           II_LineNr := 1,
                           I_Area := "STATUS_1R5".MatCard,
                           I_Map := "STATUS_BSN1".MatCard,
                           ENO => #_w1);
   IF #_w1 AND #TB1FreePosBSN THEN #TI_BSNJobNr := #CI_JobPutR34L12; END_IF;
   #TB1FreePosBSN := "MTS_MapAreaFree"(EN := NOT #TB1GripperFree AND NOT #TB1FreePosBSN,
                           II_RowNr := #TI_RowNr,
                           II_LineNr := 2,
                           I_Area := "STATUS_1R5".MatCard,
                           I_Map := "STATUS_BSN1".MatCard,
                           ENO => #_w2);
   IF #_w2 AND #TB1FreePosBSN THEN #TI_BSNJobNr := #CI_JobPutR34L23; END_IF;
   #TB1FreePosBSN := "MTS_MapAreaFree"(EN := NOT #TB1GripperFree AND NOT #TB1FreePosBSN AND ("ProdParam".BSN1_NrOfLines > 3),
                           II_RowNr := #TI_RowNr,
                           II_LineNr := 3,
                           I_Area := "STATUS_1R5".MatCard,
                           I_Map := "STATUS_BSN1".MatCard,
                           ENO => #_w3);
   IF #_w3 AND #TB1FreePosBSN THEN #TI_BSNJobNr := #CI_JobPutR34L34; END_IF;
   #TB1FreePosBSN := "MTS_MapAreaFree"(EN := NOT #TB1GripperFree AND NOT #TB1FreePosBSN AND ("ProdParam".BSN1_NrOfLines > 4),
                           II_RowNr := #TI_RowNr,
                           II_LineNr := 4,
                           I_Area := "STATUS_1R5".MatCard,
                           I_Map := "STATUS_BSN1".MatCard,
                           ENO => #_w4);
   IF #_w4 AND #TB1FreePosBSN THEN #TI_BSNJobNr := #CI_JobPutR34L45; END_IF;
   IF NOT #TB1GripperFree AND NOT #TB1FreePosBSN AND ((("ProdParam".BSN1_NrOfLines = 3) AND NOT "STATUS_BSN1".MatCard[4, 3].Occupied AND NOT "STATUS_BSN1".MatCard[3, 3].Occupied) OR (("ProdParam".BSN1_NrOfLines = 5) AND NOT "STATUS_BSN1".MatCard[4, 5].Occupied AND NOT "STATUS_BSN1".MatCard[3, 5].Occupied)) AND NOT "STATUS_BSN1".MatCard[2, 1].Occupied AND NOT "STATUS_BSN1".MatCard[1, 1].Occupied THEN
       #TI_BSNJobNr := #CI_JobPutPosX;
       #TB1FreePosBSN := TRUE;
   END_IF;
   "STATUS_BSN1".FreePosInfeed := NOT #TB1GripperFree AND #TB1FreePosBSN;
   #_w5 := NOT #TB1GripperFree AND NOT #TB1FreePosBSN;
   IF #_w5 THEN #TI_RowNr := 2; END_IF;
   #TB1FreePosBSN := "MTS_MapAreaFree"(EN := #_w5,
                           II_RowNr := #TI_RowNr,
                           II_LineNr := 1,
                           I_Area := "STATUS_1R5".MatCard,
                           I_Map := "STATUS_BSN1".MatCard,
                           ENO => #_w6);
   IF #_w6 AND #TB1FreePosBSN THEN #TI_BSNJobNr := #CI_JobPutR23L12; END_IF;
   #TB1FreePosBSN := "MTS_MapAreaFree"(EN := #_w5 AND NOT #TB1FreePosBSN,
                           II_RowNr := #TI_RowNr,
                           II_LineNr := 2,
                           I_Area := "STATUS_1R5".MatCard,
                           I_Map := "STATUS_BSN1".MatCard,
                           ENO => #_w7);
   IF #_w7 AND #TB1FreePosBSN THEN #TI_BSNJobNr := #CI_JobPutR23L23; END_IF;
   #TB1FreePosBSN := "MTS_MapAreaFree"(EN := #_w5 AND NOT #TB1FreePosBSN AND ("ProdParam".BSN1_NrOfLines > 3),
                           II_RowNr := #TI_RowNr,
                           II_LineNr := 3,
                           I_Area := "STATUS_1R5".MatCard,
                           I_Map := "STATUS_BSN1".MatCard,
                           ENO => #_w8);
   IF #_w8 AND #TB1FreePosBSN THEN #TI_BSNJobNr := #CI_JobPutR23L34; END_IF;
   #TB1FreePosBSN := "MTS_MapAreaFree"(EN := #_w5 AND NOT #TB1FreePosBSN AND ("ProdParam".BSN1_NrOfLines > 4),
                           II_RowNr := #TI_RowNr,
                           II_LineNr := 4,
                           I_Area := "STATUS_1R5".MatCard,
                           I_Map := "STATUS_BSN1".MatCard,
                           ENO => #_w9);
   IF #_w9 AND #TB1FreePosBSN THEN #TI_BSNJobNr := #CI_JobPutR23L45; END_IF;
   #_w10 := NOT #TB1GripperFree AND NOT #TB1FreePosBSN;
   IF #_w10 THEN #TI_RowNr := 1; END_IF;
   #TB1FreePosBSN := "MTS_MapAreaFree"(EN := #_w10,
                           II_RowNr := #TI_RowNr,
                           II_LineNr := 1,
                           I_Area := "STATUS_1R5".MatCard,
                           I_Map := "STATUS_BSN1".MatCard,
                           ENO => #_w11);
   IF #_w11 AND #TB1FreePosBSN THEN #TI_BSNJobNr := #CI_JobPutR12L12; END_IF;
   #TB1FreePosBSN := "MTS_MapAreaFree"(EN := #_w10 AND NOT #TB1FreePosBSN,
                           II_RowNr := #TI_RowNr,
                           II_LineNr := 2,
                           I_Area := "STATUS_1R5".MatCard,
                           I_Map := "STATUS_BSN1".MatCard,
                           ENO => #_w12);
   IF #_w12 AND #TB1FreePosBSN THEN #TI_BSNJobNr := #CI_JobPutR12L23; END_IF;
   #TB1FreePosBSN := "MTS_MapAreaFree"(EN := #_w10 AND NOT #TB1FreePosBSN AND ("ProdParam".BSN1_NrOfLines > 3),
                           II_RowNr := #TI_RowNr,
                           II_LineNr := 3,
                           I_Area := "STATUS_1R5".MatCard,
                           I_Map := "STATUS_BSN1".MatCard,
                           ENO => #_w13);
   IF #_w13 AND #TB1FreePosBSN THEN #TI_BSNJobNr := #CI_JobPutR12L34; END_IF;
   #TB1FreePosBSN := "MTS_MapAreaFree"(EN := #_w10 AND NOT #TB1FreePosBSN AND ("ProdParam".BSN1_NrOfLines > 4),
                           II_RowNr := #TI_RowNr,
                           II_LineNr := 4,
                           I_Area := "STATUS_1R5".MatCard,
                           I_Map := "STATUS_BSN1".MatCard,
                           ENO => #_w14);
   IF #_w14 AND #TB1FreePosBSN THEN #TI_BSNJobNr := #CI_JobPutR12L45; END_IF;
END_REGION

REGION Network 25: Robot RO01 - BSN1 - put command
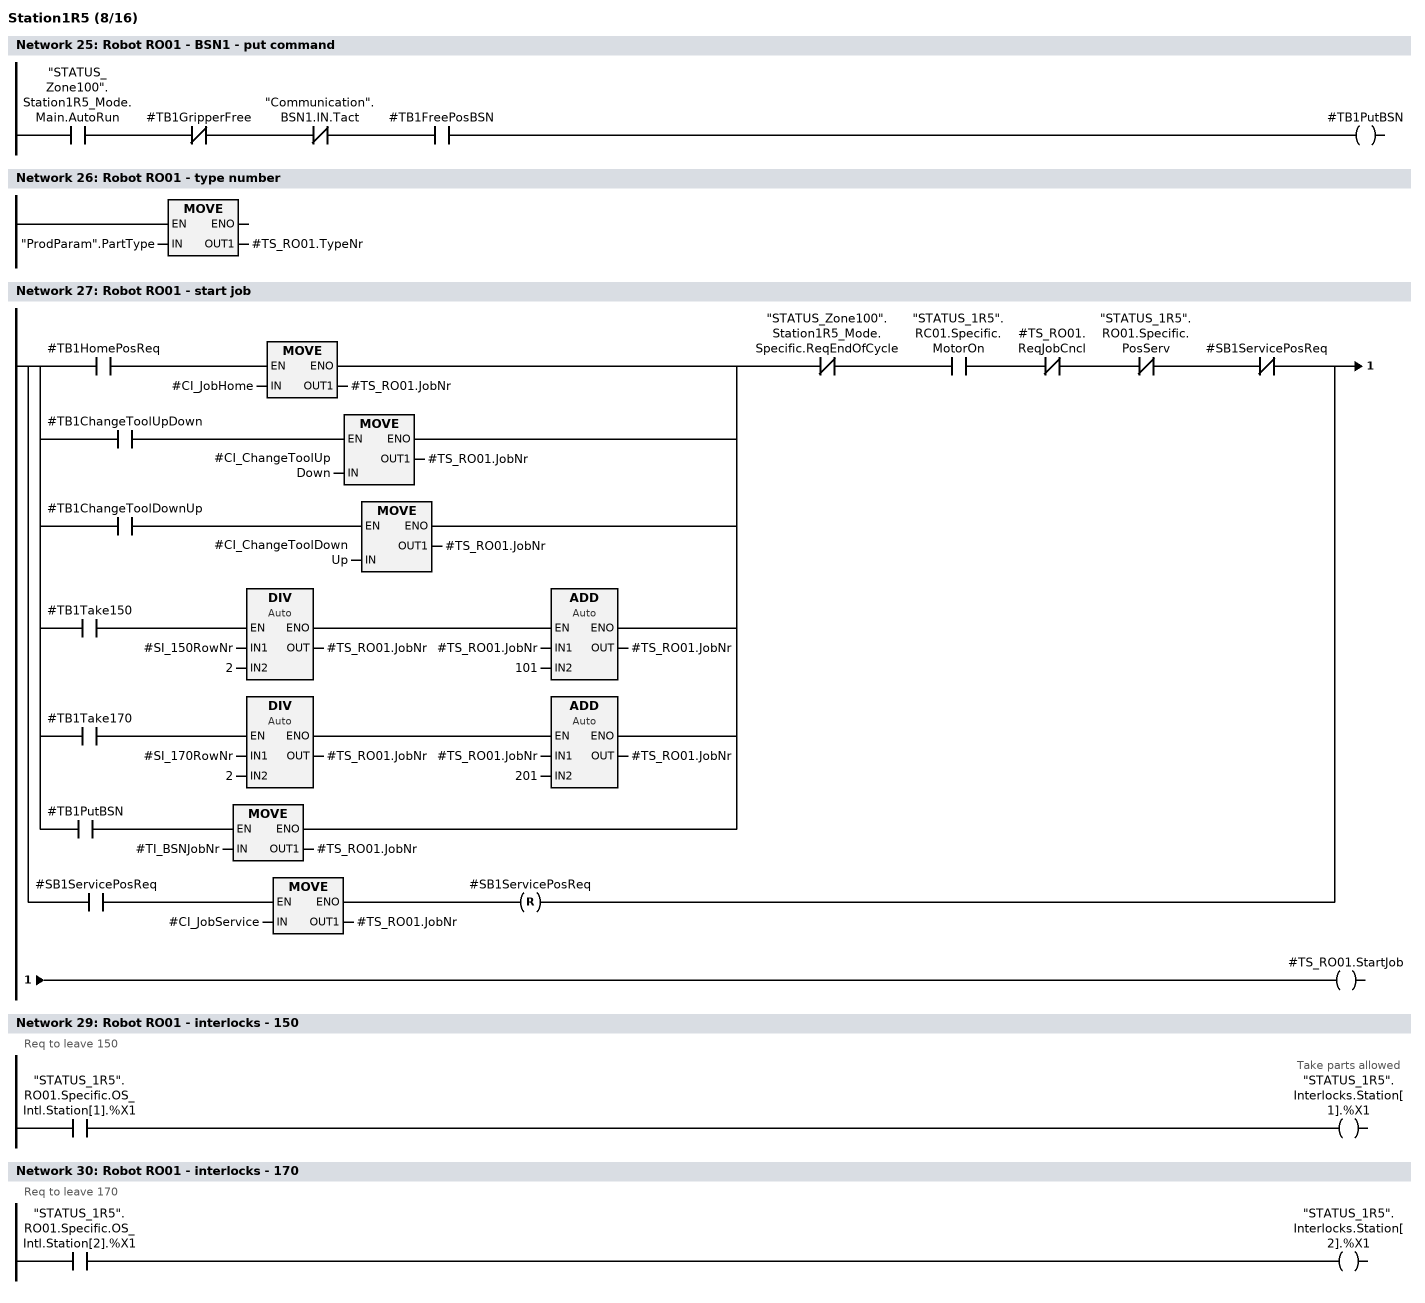
   RUNG wire#powerrail
      Contact( "STATUS_Zone100".Station1R5_Mode.Main.AutoRun )
      I_Contact( #TB1GripperFree )
      I_Contact( "Communication".BSN1.IN.Tact )
      Contact( #TB1FreePosBSN )
      Coil( #TB1PutBSN )
   END_RUNG
   // the same network as SCL:
   #TB1PutBSN := "STATUS_Zone100".Station1R5_Mode.Main.AutoRun AND NOT #TB1GripperFree AND NOT "Communication".BSN1.IN.Tact AND #TB1FreePosBSN;
END_REGION

REGION Network 26: Robot RO01 - type number
   RUNG wire#powerrail
      Move(in := "ProdParam".PartType, out1 => #TS_RO01.TypeNr)
   END_RUNG
   // the same network as SCL:
   #TS_RO01.TypeNr := "ProdParam".PartType;
END_REGION

REGION Network 27: Robot RO01 - start job
   RUNG wire#powerrail
      Contact( #TB1HomePosReq )
      Move(in := #CI_JobHome, out1 => #TS_RO01.JobNr)
      wire#w1
      I_Contact( "STATUS_Zone100".Station1R5_Mode.Specific.ReqEndOfCycle )
      Contact( "STATUS_1R5".RC01.Specific.MotorOn )
      I_Contact( #TS_RO01.ReqJobCncl )
      I_Contact( "STATUS_1R5".RO01.Specific.PosServ )
      I_Contact( #SB1ServicePosReq )
      wire#w2
      Coil( #TS_RO01.StartJob )
   END_RUNG
   RUNG wire#powerrail
      Contact( #TB1ChangeToolUpDown )
      Move(in := #CI_ChangeToolUpDown, out1 => #TS_RO01.JobNr)
   END_RUNG wire#w1
   RUNG wire#powerrail
      Contact( #TB1ChangeToolDownUp )
      Move(in := #CI_ChangeToolDownUp, out1 => #TS_RO01.JobNr)
   END_RUNG wire#w1
   RUNG wire#powerrail
      Contact( #TB1Take150 )
      Div(in1 := #SI_150RowNr, in2 := 2, out => #TS_RO01.JobNr)
      Add(in1 := #TS_RO01.JobNr, in2 := 101, out => #TS_RO01.JobNr)
   END_RUNG wire#w1
   RUNG wire#powerrail
      Contact( #TB1Take170 )
      Div(in1 := #SI_170RowNr, in2 := 2, out => #TS_RO01.JobNr)
      Add(in1 := #TS_RO01.JobNr, in2 := 201, out => #TS_RO01.JobNr)
   END_RUNG wire#w1
   RUNG wire#powerrail
      Contact( #TB1PutBSN )
      Move(in := #TI_BSNJobNr, out1 => #TS_RO01.JobNr)
   END_RUNG wire#w1
   RUNG wire#powerrail
      Contact( #SB1ServicePosReq )
      Move(in := #CI_JobService, out1 => #TS_RO01.JobNr)
      R_Coil( #SB1ServicePosReq )
   END_RUNG wire#w2
   // the same network as SCL:
   IF #TB1HomePosReq THEN #TS_RO01.JobNr := #CI_JobHome; END_IF;
   IF #TB1ChangeToolUpDown THEN #TS_RO01.JobNr := #CI_ChangeToolUpDown; END_IF;
   IF #TB1ChangeToolDownUp THEN #TS_RO01.JobNr := #CI_ChangeToolDownUp; END_IF;
   IF #TB1Take150 THEN
       #TS_RO01.JobNr := #SI_150RowNr / 2;
       #TS_RO01.JobNr := #TS_RO01.JobNr + 101;
   END_IF;
   IF #TB1Take170 THEN
       #TS_RO01.JobNr := #SI_170RowNr / 2;
       #TS_RO01.JobNr := #TS_RO01.JobNr + 201;
   END_IF;
   IF #TB1PutBSN THEN #TS_RO01.JobNr := #TI_BSNJobNr; END_IF;
   IF #SB1ServicePosReq THEN #TS_RO01.JobNr := #CI_JobService; END_IF;
   #_w1 := #SB1ServicePosReq;
   #_w2 := (#TB1HomePosReq OR #TB1ChangeToolUpDown OR #TB1ChangeToolDownUp OR #TB1Take150 OR #TB1Take170 OR #TB1PutBSN) AND NOT "STATUS_Zone100".Station1R5_Mode.Specific.ReqEndOfCycle AND "STATUS_1R5".RC01.Specific.MotorOn AND NOT #TS_RO01.ReqJobCncl AND NOT "STATUS_1R5".RO01.Specific.PosServ AND NOT #SB1ServicePosReq;
   IF #_w1 THEN #SB1ServicePosReq := FALSE; END_IF;
   #TS_RO01.StartJob := #_w2 OR #_w1;
END_REGION

REGION Network 28: *************** Interlocks ***************
END_REGION

REGION Network 29: Robot RO01 - interlocks - 150
   // Req to leave 150
   RUNG wire#powerrail
      Contact( "STATUS_1R5".RO01.Specific.OS_Intl.Station[1].%X1 )
      Coil( "STATUS_1R5".Interlocks.Station[1].%X1 )   // Take parts allowed
   END_RUNG
   // the same network as SCL:
   "STATUS_1R5".Interlocks.Station[1].%X1 := "STATUS_1R5".RO01.Specific.OS_Intl.Station[1].%X1;   // Take parts allowed
END_REGION

REGION Network 30: Robot RO01 - interlocks - 170
   // Req to leave 170
   RUNG wire#powerrail
      Contact( "STATUS_1R5".RO01.Specific.OS_Intl.Station[2].%X1 )
      Coil( "STATUS_1R5".Interlocks.Station[2].%X1 )
   END_RUNG
   // the same network as SCL:
   "STATUS_1R5".Interlocks.Station[2].%X1 := "STATUS_1R5".RO01.Specific.OS_Intl.Station[2].%X1;
END_REGION

REGION Network 31: Robot RO01 - interlocks - BSN1
   // Req to leave BSN1
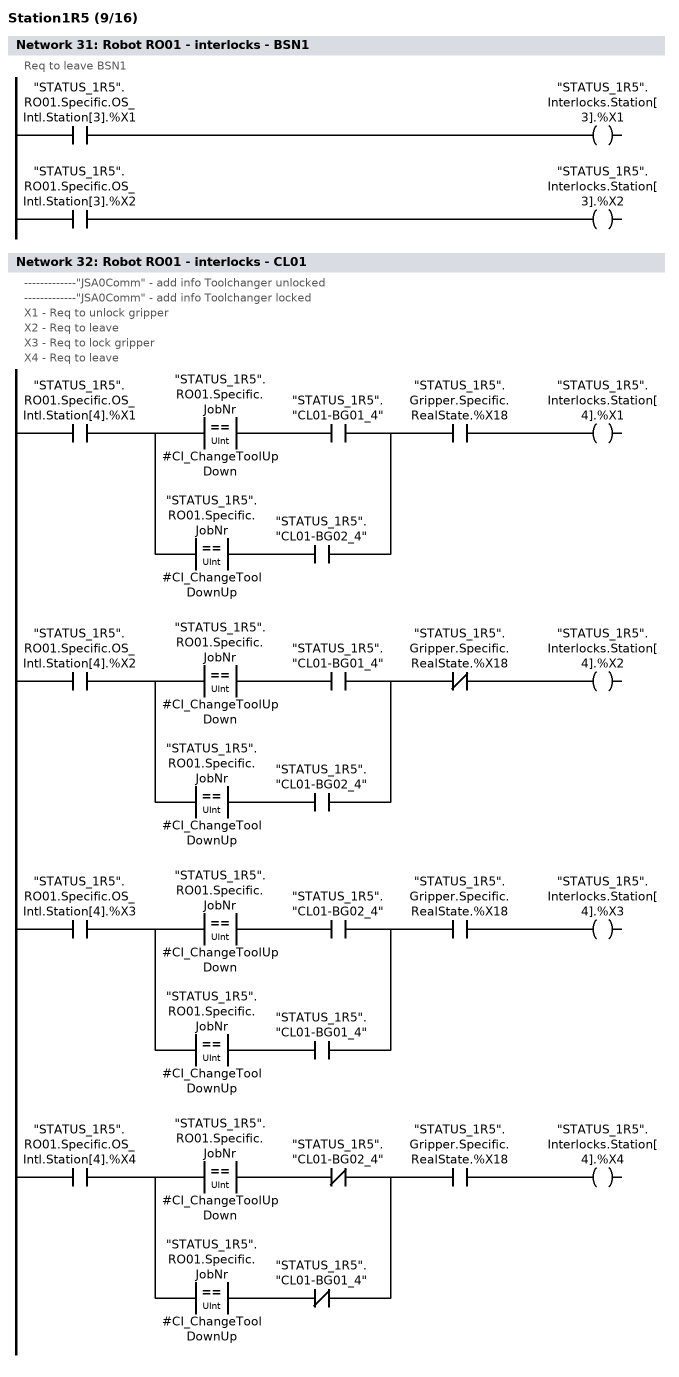
   RUNG wire#powerrail
      Contact( "STATUS_1R5".RO01.Specific.OS_Intl.Station[3].%X1 )
      Coil( "STATUS_1R5".Interlocks.Station[3].%X1 )
   END_RUNG
   RUNG wire#powerrail
      Contact( "STATUS_1R5".RO01.Specific.OS_Intl.Station[3].%X2 )
      Coil( "STATUS_1R5".Interlocks.Station[3].%X2 )
   END_RUNG
   // the same network as SCL:
   "STATUS_1R5".Interlocks.Station[3].%X1 := "STATUS_1R5".RO01.Specific.OS_Intl.Station[3].%X1;
   "STATUS_1R5".Interlocks.Station[3].%X2 := "STATUS_1R5".RO01.Specific.OS_Intl.Station[3].%X2;
END_REGION

REGION Network 32: Robot RO01 - interlocks - CL01
   // -------------"JSA0Comm" - add info Toolchanger unlocked
   // -------------"JSA0Comm" - add info Toolchanger locked
   // 
   // 
   // X1 - Req to unlock gripper
   // X2 - Req to leave
   // X3 - Req to lock gripper
   // X4 - Req to leave
   RUNG wire#powerrail
      Contact( "STATUS_1R5".RO01.Specific.OS_Intl.Station[4].%X1 )
      wire#w1
      { S7_Templates := "SrcType := UInt" } EQ_Contact(in1 := "STATUS_1R5".RO01.Specific.JobNr, in2 := #CI_ChangeToolUpDown)
      Contact( "STATUS_1R5"."CL01-BG01_4" )
      wire#w2
      Contact( "STATUS_1R5".Gripper.Specific.RealState.%X18 )
      Coil( "STATUS_1R5".Interlocks.Station[4].%X1 )
   END_RUNG
   RUNG wire#w1
      { S7_Templates := "SrcType := UInt" } EQ_Contact(in1 := "STATUS_1R5".RO01.Specific.JobNr, in2 := #CI_ChangeToolDownUp)
      Contact( "STATUS_1R5"."CL01-BG02_4" )
   END_RUNG wire#w2
   RUNG wire#powerrail
      Contact( "STATUS_1R5".RO01.Specific.OS_Intl.Station[4].%X2 )
      wire#w3
      { S7_Templates := "SrcType := UInt" } EQ_Contact(in1 := "STATUS_1R5".RO01.Specific.JobNr, in2 := #CI_ChangeToolUpDown)
      Contact( "STATUS_1R5"."CL01-BG01_4" )
      wire#w4
      I_Contact( "STATUS_1R5".Gripper.Specific.RealState.%X18 )
      Coil( "STATUS_1R5".Interlocks.Station[4].%X2 )
   END_RUNG
   RUNG wire#w3
      { S7_Templates := "SrcType := UInt" } EQ_Contact(in1 := "STATUS_1R5".RO01.Specific.JobNr, in2 := #CI_ChangeToolDownUp)
      Contact( "STATUS_1R5"."CL01-BG02_4" )
   END_RUNG wire#w4
   RUNG wire#powerrail
      Contact( "STATUS_1R5".RO01.Specific.OS_Intl.Station[4].%X3 )
      wire#w5
      { S7_Templates := "SrcType := UInt" } EQ_Contact(in1 := "STATUS_1R5".RO01.Specific.JobNr, in2 := #CI_ChangeToolUpDown)
      Contact( "STATUS_1R5"."CL01-BG02_4" )
      wire#w6
      Contact( "STATUS_1R5".Gripper.Specific.RealState.%X18 )
      Coil( "STATUS_1R5".Interlocks.Station[4].%X3 )
   END_RUNG
   RUNG wire#w5
      { S7_Templates := "SrcType := UInt" } EQ_Contact(in1 := "STATUS_1R5".RO01.Specific.JobNr, in2 := #CI_ChangeToolDownUp)
      Contact( "STATUS_1R5"."CL01-BG01_4" )
   END_RUNG wire#w6
   RUNG wire#powerrail
      Contact( "STATUS_1R5".RO01.Specific.OS_Intl.Station[4].%X4 )
      wire#w7
      { S7_Templates := "SrcType := UInt" } EQ_Contact(in1 := "STATUS_1R5".RO01.Specific.JobNr, in2 := #CI_ChangeToolUpDown)
      I_Contact( "STATUS_1R5"."CL01-BG02_4" )
      wire#w8
      Contact( "STATUS_1R5".Gripper.Specific.RealState.%X18 )
      Coil( "STATUS_1R5".Interlocks.Station[4].%X4 )
   END_RUNG
   RUNG wire#w7
      { S7_Templates := "SrcType := UInt" } EQ_Contact(in1 := "STATUS_1R5".RO01.Specific.JobNr, in2 := #CI_ChangeToolDownUp)
      I_Contact( "STATUS_1R5"."CL01-BG01_4" )
   END_RUNG wire#w8
   // the same network as SCL:
   "STATUS_1R5".Interlocks.Station[4].%X1 := "STATUS_1R5".RO01.Specific.OS_Intl.Station[4].%X1 AND ((("STATUS_1R5".RO01.Specific.JobNr = #CI_ChangeToolUpDown) AND "STATUS_1R5"."CL01-BG01_4") OR (("STATUS_1R5".RO01.Specific.JobNr = #CI_ChangeToolDownUp) AND "STATUS_1R5"."CL01-BG02_4")) AND "STATUS_1R5".Gripper.Specific.RealState.%X18;
   "STATUS_1R5".Interlocks.Station[4].%X2 := "STATUS_1R5".RO01.Specific.OS_Intl.Station[4].%X2 AND ((("STATUS_1R5".RO01.Specific.JobNr = #CI_ChangeToolUpDown) AND "STATUS_1R5"."CL01-BG01_4") OR (("STATUS_1R5".RO01.Specific.JobNr = #CI_ChangeToolDownUp) AND "STATUS_1R5"."CL01-BG02_4")) AND NOT "STATUS_1R5".Gripper.Specific.RealState.%X18;
   "STATUS_1R5".Interlocks.Station[4].%X3 := "STATUS_1R5".RO01.Specific.OS_Intl.Station[4].%X3 AND ((("STATUS_1R5".RO01.Specific.JobNr = #CI_ChangeToolUpDown) AND "STATUS_1R5"."CL01-BG02_4") OR (("STATUS_1R5".RO01.Specific.JobNr = #CI_ChangeToolDownUp) AND "STATUS_1R5"."CL01-BG01_4")) AND "STATUS_1R5".Gripper.Specific.RealState.%X18;
   "STATUS_1R5".Interlocks.Station[4].%X4 := "STATUS_1R5".RO01.Specific.OS_Intl.Station[4].%X4 AND ((("STATUS_1R5".RO01.Specific.JobNr = #CI_ChangeToolUpDown) AND NOT "STATUS_1R5"."CL01-BG02_4") OR (("STATUS_1R5".RO01.Specific.JobNr = #CI_ChangeToolDownUp) AND NOT "STATUS_1R5"."CL01-BG01_4")) AND "STATUS_1R5".Gripper.Specific.RealState.%X18;
END_REGION

REGION Network 33: *************** Zone releases ***************
END_REGION

REGION Network 34: Robot RO01 - zone 1 release - 150 - evaluation in FB Station150
END_REGION

REGION Network 35: Robot RO01 - zone 2 release - 170 - evaluation in FB Station170
END_REGION

REGION Network 36: Robot RO01 - zone 3 release - BSN1 - evaluation in FB StationBSN1
END_REGION

REGION Network 37: Robot RO01 - zone 4 release - CL01
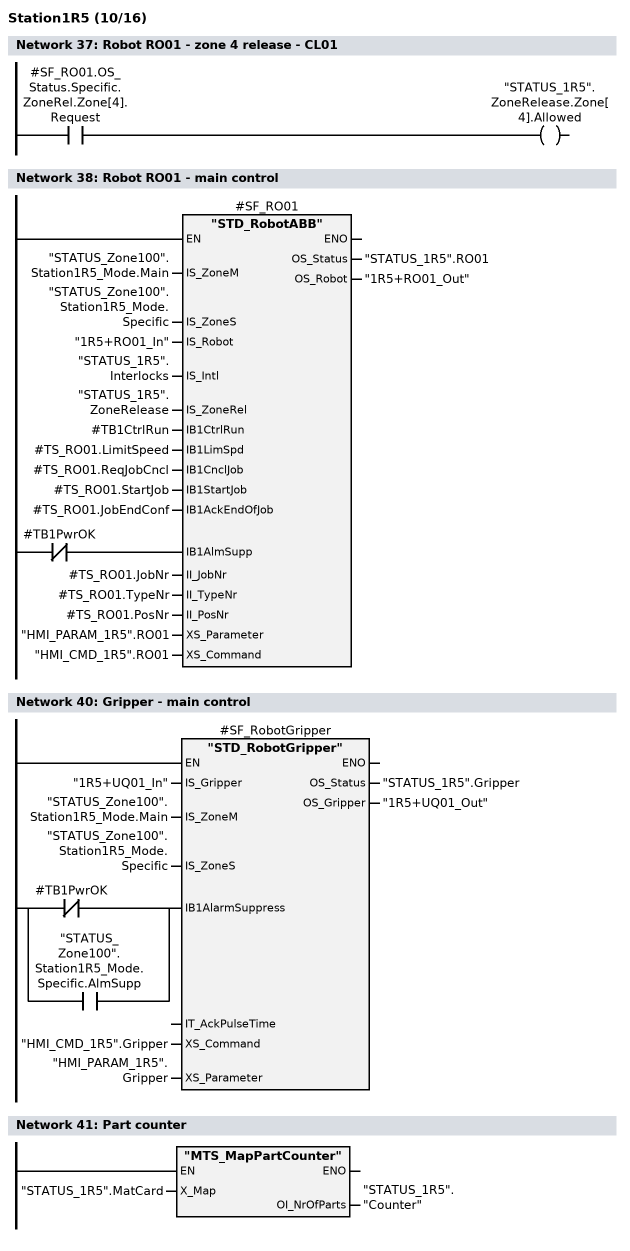
   RUNG wire#powerrail
      Contact( #SF_RO01.OS_Status.Specific.ZoneRel.Zone[4].Request )
      Coil( "STATUS_1R5".ZoneRelease.Zone[4].Allowed )
   END_RUNG
   // the same network as SCL:
   "STATUS_1R5".ZoneRelease.Zone[4].Allowed := #SF_RO01.OS_Status.Specific.ZoneRel.Zone[4].Request;
END_REGION

REGION Network 38: Robot RO01 - main control
   RUNG wire#powerrail
      #SF_RO01(IB1AlmSupp := wire#w1, IS_ZoneM := "STATUS_Zone100".Station1R5_Mode.Main, IS_ZoneS := "STATUS_Zone100".Station1R5_Mode.Specific, IS_Robot := "1R5+RO01_In", IS_Intl := "STATUS_1R5".Interlocks, IS_ZoneRel := "STATUS_1R5".ZoneRelease, IB1CtrlRun := #TB1CtrlRun, IB1LimSpd := #TS_RO01.LimitSpeed, IB1CnclJob := #TS_RO01.ReqJobCncl, IB1StartJob := #TS_RO01.StartJob, IB1AckEndOfJob := #TS_RO01.JobEndConf, II_JobNr := #TS_RO01.JobNr, II_TypeNr := #TS_RO01.TypeNr, II_PosNr := #TS_RO01.PosNr, XS_Parameter := "HMI_PARAM_1R5".RO01, XS_Command := "HMI_CMD_1R5".RO01, OS_Status => "STATUS_1R5".RO01, OS_Robot => "1R5+RO01_Out")
   END_RUNG
   RUNG wire#powerrail
      I_Contact( #TB1PwrOK )
   END_RUNG wire#w1
   // the same network as SCL:
   #SF_RO01(IS_ZoneM := "STATUS_Zone100".Station1R5_Mode.Main,   // "STD_RobotABB"
            IS_ZoneS := "STATUS_Zone100".Station1R5_Mode.Specific,
            IS_Robot := "1R5+RO01_In",
            IS_Intl := "STATUS_1R5".Interlocks,
            IS_ZoneRel := "STATUS_1R5".ZoneRelease,
            IB1CtrlRun := #TB1CtrlRun,
            IB1LimSpd := #TS_RO01.LimitSpeed,
            IB1CnclJob := #TS_RO01.ReqJobCncl,
            IB1StartJob := #TS_RO01.StartJob,
            IB1AckEndOfJob := #TS_RO01.JobEndConf,
            IB1AlmSupp := NOT #TB1PwrOK,
            II_JobNr := #TS_RO01.JobNr,
            II_TypeNr := #TS_RO01.TypeNr,
            II_PosNr := #TS_RO01.PosNr,
            XS_Parameter := "HMI_PARAM_1R5".RO01,
            XS_Command := "HMI_CMD_1R5".RO01,
            OS_Status => "STATUS_1R5".RO01,
            OS_Robot => "1R5+RO01_Out");
END_REGION

REGION Network 39: *************** Gripper ***************
END_REGION

REGION Network 40: Gripper - main control
   RUNG wire#powerrail
      #SF_RobotGripper(IB1AlarmSuppress := wire#w1, IS_Gripper := "1R5+UQ01_In", IS_ZoneM := "STATUS_Zone100".Station1R5_Mode.Main, IS_ZoneS := "STATUS_Zone100".Station1R5_Mode.Specific, IT_AckPulseTime :=, XS_Command := "HMI_CMD_1R5".Gripper, XS_Parameter := "HMI_PARAM_1R5".Gripper, OS_Status => "STATUS_1R5".Gripper, OS_Gripper => "1R5+UQ01_Out")
   END_RUNG
   RUNG wire#powerrail
      I_Contact( #TB1PwrOK )
   END_RUNG wire#w1
   RUNG wire#powerrail
      Contact( "STATUS_Zone100".Station1R5_Mode.Specific.AlmSupp )
   END_RUNG wire#w1
   // the same network as SCL:
   #SF_RobotGripper(IS_Gripper := "1R5+UQ01_In",   // "STD_RobotGripper"
                    IS_ZoneM := "STATUS_Zone100".Station1R5_Mode.Main,
                    IS_ZoneS := "STATUS_Zone100".Station1R5_Mode.Specific,
                    IB1AlarmSuppress := NOT #TB1PwrOK OR "STATUS_Zone100".Station1R5_Mode.Specific.AlmSupp,
                    XS_Command := "HMI_CMD_1R5".Gripper,
                    XS_Parameter := "HMI_PARAM_1R5".Gripper,
                    OS_Status => "STATUS_1R5".Gripper,
                    OS_Gripper => "1R5+UQ01_Out");
END_REGION

REGION Network 41: Part counter
   RUNG wire#powerrail
      "MTS_MapPartCounter"(X_Map := "STATUS_1R5".MatCard, OI_NrOfParts => "STATUS_1R5"."Counter")
   END_RUNG
   // the same network as SCL:
   "MTS_MapPartCounter"(X_Map := "STATUS_1R5".MatCard, OI_NrOfParts => "STATUS_1R5"."Counter");
END_REGION

REGION Network 42: *************** Material flow ***************
END_REGION

REGION Network 43: Clear positions and map - commands
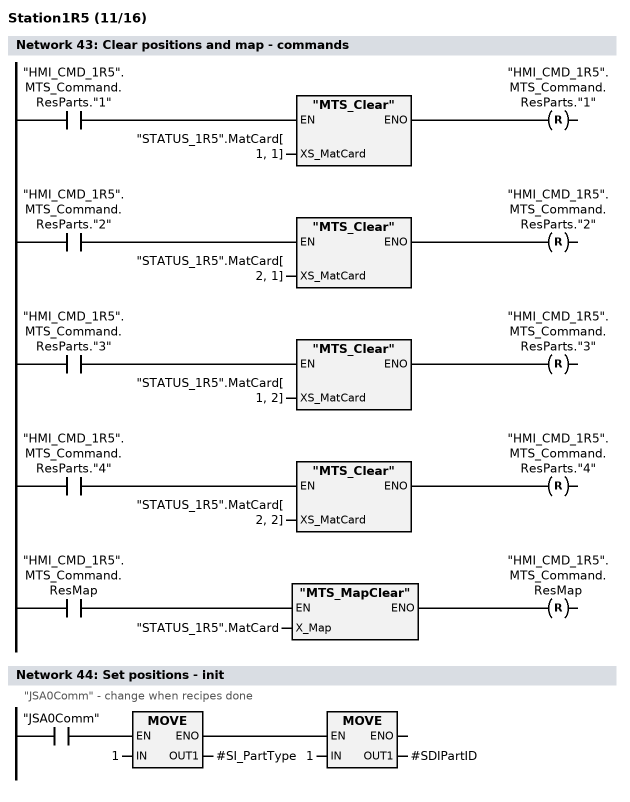
   RUNG wire#powerrail
      Contact( "HMI_CMD_1R5".MTS_Command.ResParts."1" )
      "MTS_Clear"(XS_MatCard := "STATUS_1R5".MatCard[1, 1])
      R_Coil( "HMI_CMD_1R5".MTS_Command.ResParts."1" )
   END_RUNG
   RUNG wire#powerrail
      Contact( "HMI_CMD_1R5".MTS_Command.ResParts."2" )
      "MTS_Clear"(XS_MatCard := "STATUS_1R5".MatCard[2, 1])
      R_Coil( "HMI_CMD_1R5".MTS_Command.ResParts."2" )
   END_RUNG
   RUNG wire#powerrail
      Contact( "HMI_CMD_1R5".MTS_Command.ResParts."3" )
      "MTS_Clear"(XS_MatCard := "STATUS_1R5".MatCard[1, 2])
      R_Coil( "HMI_CMD_1R5".MTS_Command.ResParts."3" )
   END_RUNG
   RUNG wire#powerrail
      Contact( "HMI_CMD_1R5".MTS_Command.ResParts."4" )
      "MTS_Clear"(XS_MatCard := "STATUS_1R5".MatCard[2, 2])
      R_Coil( "HMI_CMD_1R5".MTS_Command.ResParts."4" )
   END_RUNG
   RUNG wire#powerrail
      Contact( "HMI_CMD_1R5".MTS_Command.ResMap )
      "MTS_MapClear"(X_Map := "STATUS_1R5".MatCard)
      R_Coil( "HMI_CMD_1R5".MTS_Command.ResMap )
   END_RUNG
   // the same network as SCL:
   "MTS_Clear"(EN := "HMI_CMD_1R5".MTS_Command.ResParts."1",
               XS_MatCard := "STATUS_1R5".MatCard[1, 1],
               ENO => #_w1);
   IF #_w1 THEN "HMI_CMD_1R5".MTS_Command.ResParts."1" := FALSE; END_IF;
   "MTS_Clear"(EN := "HMI_CMD_1R5".MTS_Command.ResParts."2",
               XS_MatCard := "STATUS_1R5".MatCard[2, 1],
               ENO => #_w2);
   IF #_w2 THEN "HMI_CMD_1R5".MTS_Command.ResParts."2" := FALSE; END_IF;
   "MTS_Clear"(EN := "HMI_CMD_1R5".MTS_Command.ResParts."3",
               XS_MatCard := "STATUS_1R5".MatCard[1, 2],
               ENO => #_w3);
   IF #_w3 THEN "HMI_CMD_1R5".MTS_Command.ResParts."3" := FALSE; END_IF;
   "MTS_Clear"(EN := "HMI_CMD_1R5".MTS_Command.ResParts."4",
               XS_MatCard := "STATUS_1R5".MatCard[2, 2],
               ENO => #_w4);
   IF #_w4 THEN "HMI_CMD_1R5".MTS_Command.ResParts."4" := FALSE; END_IF;
   "MTS_MapClear"(EN := "HMI_CMD_1R5".MTS_Command.ResMap, X_Map := "STATUS_1R5".MatCard, ENO => #_w5);
   IF #_w5 THEN "HMI_CMD_1R5".MTS_Command.ResMap := FALSE; END_IF;
END_REGION

REGION Network 44: Set positions - init
   // "JSA0Comm" - change when recipes done
   RUNG wire#powerrail
      Contact( "JSA0Comm" )
      Move(in := 1, out1 => #SI_PartType)
      Move(in := 1, out1 => #SDIPartID)
   END_RUNG
   // the same network as SCL:
   IF "JSA0Comm" THEN
       #SI_PartType := 1;
       #SDIPartID := 1;
   END_IF;
END_REGION

REGION Network 45: Set positions and map - commands
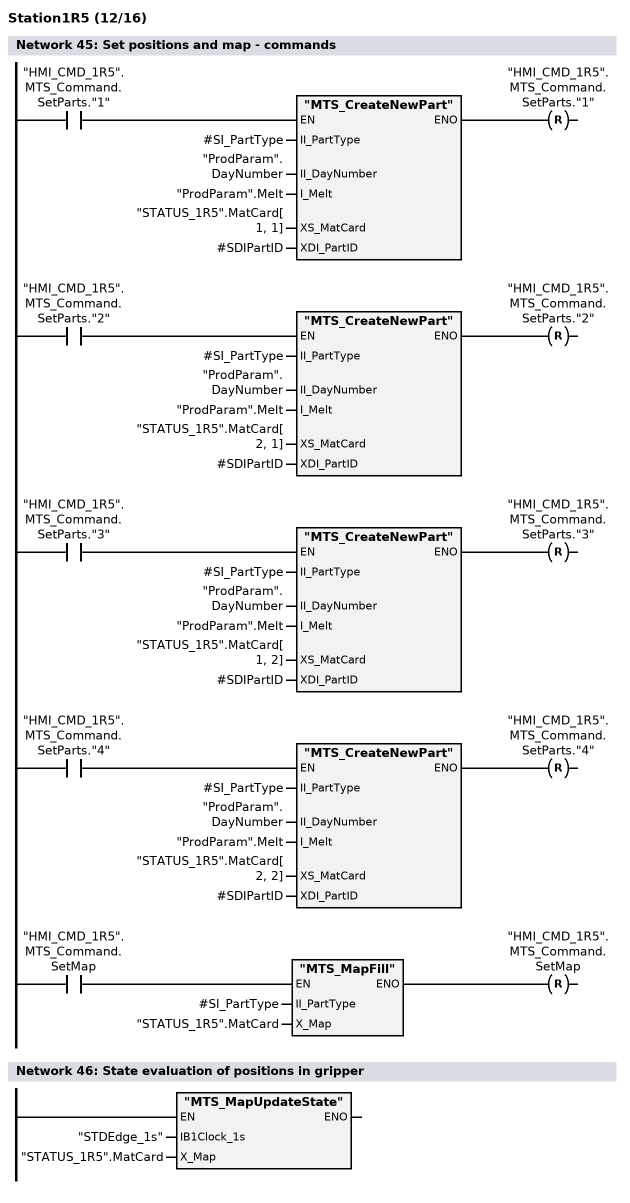
   RUNG wire#powerrail
      Contact( "HMI_CMD_1R5".MTS_Command.SetParts."1" )
      "MTS_CreateNewPart"(II_PartType := #SI_PartType, II_DayNumber := "ProdParam".DayNumber, I_Melt := "ProdParam".Melt, XS_MatCard := "STATUS_1R5".MatCard[1, 1], XDI_PartID := #SDIPartID)
      R_Coil( "HMI_CMD_1R5".MTS_Command.SetParts."1" )
   END_RUNG
   RUNG wire#powerrail
      Contact( "HMI_CMD_1R5".MTS_Command.SetParts."2" )
      "MTS_CreateNewPart"(II_PartType := #SI_PartType, II_DayNumber := "ProdParam".DayNumber, I_Melt := "ProdParam".Melt, XS_MatCard := "STATUS_1R5".MatCard[2, 1], XDI_PartID := #SDIPartID)
      R_Coil( "HMI_CMD_1R5".MTS_Command.SetParts."2" )
   END_RUNG
   RUNG wire#powerrail
      Contact( "HMI_CMD_1R5".MTS_Command.SetParts."3" )
      "MTS_CreateNewPart"(II_PartType := #SI_PartType, II_DayNumber := "ProdParam".DayNumber, I_Melt := "ProdParam".Melt, XS_MatCard := "STATUS_1R5".MatCard[1, 2], XDI_PartID := #SDIPartID)
      R_Coil( "HMI_CMD_1R5".MTS_Command.SetParts."3" )
   END_RUNG
   RUNG wire#powerrail
      Contact( "HMI_CMD_1R5".MTS_Command.SetParts."4" )
      "MTS_CreateNewPart"(II_PartType := #SI_PartType, II_DayNumber := "ProdParam".DayNumber, I_Melt := "ProdParam".Melt, XS_MatCard := "STATUS_1R5".MatCard[2, 2], XDI_PartID := #SDIPartID)
      R_Coil( "HMI_CMD_1R5".MTS_Command.SetParts."4" )
   END_RUNG
   RUNG wire#powerrail
      Contact( "HMI_CMD_1R5".MTS_Command.SetMap )
      "MTS_MapFill"(II_PartType := #SI_PartType, X_Map := "STATUS_1R5".MatCard)
      R_Coil( "HMI_CMD_1R5".MTS_Command.SetMap )
   END_RUNG
   // the same network as SCL:
   "MTS_CreateNewPart"(EN := "HMI_CMD_1R5".MTS_Command.SetParts."1",
                       II_PartType := #SI_PartType,
                       II_DayNumber := "ProdParam".DayNumber,
                       I_Melt := "ProdParam".Melt,
                       XS_MatCard := "STATUS_1R5".MatCard[1, 1],
                       XDI_PartID := #SDIPartID,
                       ENO => #_w1);
   IF #_w1 THEN "HMI_CMD_1R5".MTS_Command.SetParts."1" := FALSE; END_IF;
   "MTS_CreateNewPart"(EN := "HMI_CMD_1R5".MTS_Command.SetParts."2",
                       II_PartType := #SI_PartType,
                       II_DayNumber := "ProdParam".DayNumber,
                       I_Melt := "ProdParam".Melt,
                       XS_MatCard := "STATUS_1R5".MatCard[2, 1],
                       XDI_PartID := #SDIPartID,
                       ENO => #_w2);
   IF #_w2 THEN "HMI_CMD_1R5".MTS_Command.SetParts."2" := FALSE; END_IF;
   "MTS_CreateNewPart"(EN := "HMI_CMD_1R5".MTS_Command.SetParts."3",
                       II_PartType := #SI_PartType,
                       II_DayNumber := "ProdParam".DayNumber,
                       I_Melt := "ProdParam".Melt,
                       XS_MatCard := "STATUS_1R5".MatCard[1, 2],
                       XDI_PartID := #SDIPartID,
                       ENO => #_w3);
   IF #_w3 THEN "HMI_CMD_1R5".MTS_Command.SetParts."3" := FALSE; END_IF;
   "MTS_CreateNewPart"(EN := "HMI_CMD_1R5".MTS_Command.SetParts."4",
                       II_PartType := #SI_PartType,
                       II_DayNumber := "ProdParam".DayNumber,
                       I_Melt := "ProdParam".Melt,
                       XS_MatCard := "STATUS_1R5".MatCard[2, 2],
                       XDI_PartID := #SDIPartID,
                       ENO => #_w4);
   IF #_w4 THEN "HMI_CMD_1R5".MTS_Command.SetParts."4" := FALSE; END_IF;
   "MTS_MapFill"(EN := "HMI_CMD_1R5".MTS_Command.SetMap,
                 II_PartType := #SI_PartType,
                 X_Map := "STATUS_1R5".MatCard,
                 ENO => #_w5);
   IF #_w5 THEN "HMI_CMD_1R5".MTS_Command.SetMap := FALSE; END_IF;
END_REGION

REGION Network 46: State evaluation of positions in gripper
   RUNG wire#powerrail
      "MTS_MapUpdateState"(IB1Clock_1s := "STDEdge_1s", X_Map := "STATUS_1R5".MatCard)
   END_RUNG
   // the same network as SCL:
   "MTS_MapUpdateState"(IB1Clock_1s := "STDEdge_1s", X_Map := "STATUS_1R5".MatCard);
END_REGION

REGION Network 47: Data transfer: 150/170 - row number
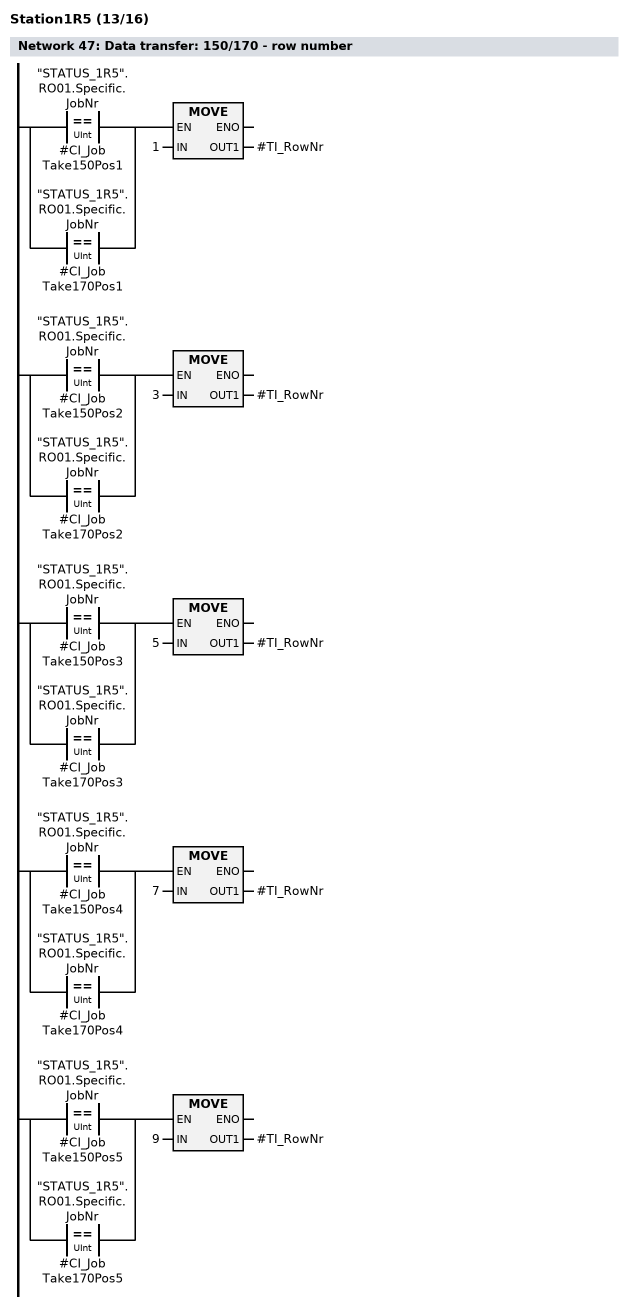
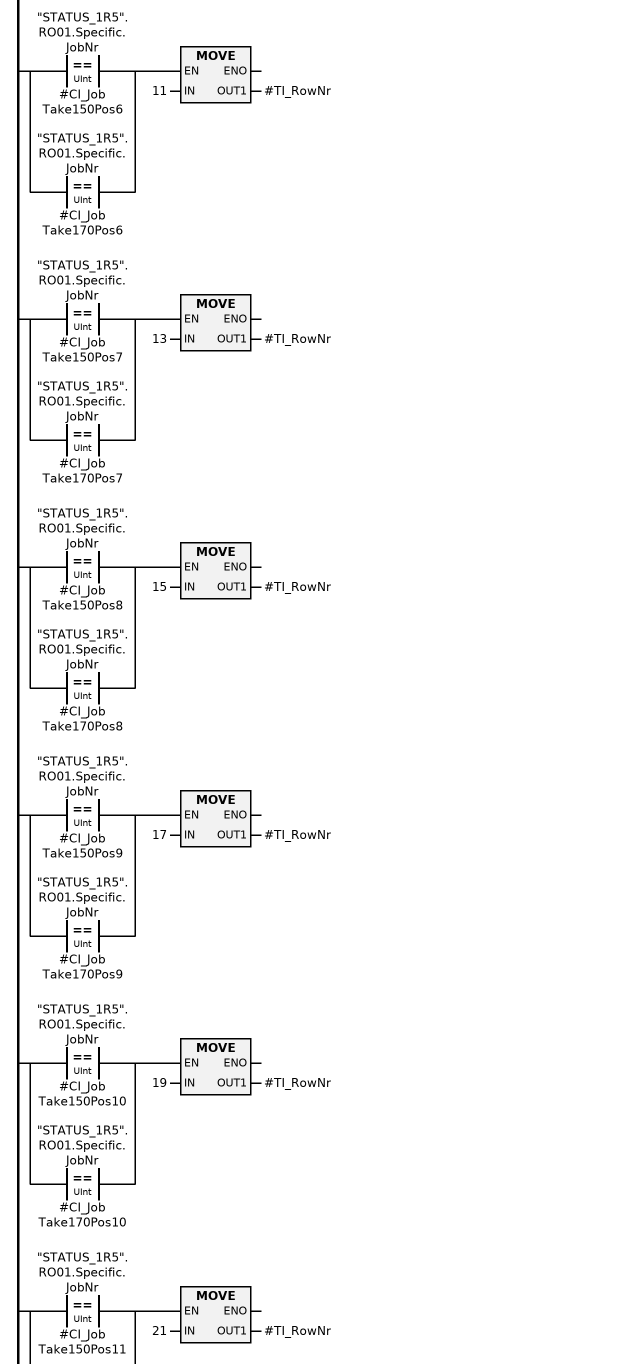
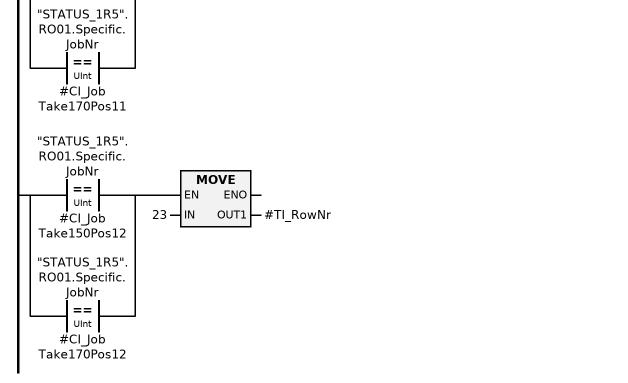
   RUNG wire#powerrail
      { S7_Templates := "SrcType := UInt" } EQ_Contact(in1 := "STATUS_1R5".RO01.Specific.JobNr, in2 := #CI_JobTake150Pos1)
      wire#w1
      Move(in := 1, out1 => #TI_RowNr)
   END_RUNG
   RUNG wire#powerrail
      { S7_Templates := "SrcType := UInt" } EQ_Contact(in1 := "STATUS_1R5".RO01.Specific.JobNr, in2 := #CI_JobTake170Pos1)
   END_RUNG wire#w1
   RUNG wire#powerrail
      { S7_Templates := "SrcType := UInt" } EQ_Contact(in1 := "STATUS_1R5".RO01.Specific.JobNr, in2 := #CI_JobTake150Pos2)
      wire#w2
      Move(in := 3, out1 => #TI_RowNr)
   END_RUNG
   RUNG wire#powerrail
      { S7_Templates := "SrcType := UInt" } EQ_Contact(in1 := "STATUS_1R5".RO01.Specific.JobNr, in2 := #CI_JobTake170Pos2)
   END_RUNG wire#w2
   RUNG wire#powerrail
      { S7_Templates := "SrcType := UInt" } EQ_Contact(in1 := "STATUS_1R5".RO01.Specific.JobNr, in2 := #CI_JobTake150Pos3)
      wire#w3
      Move(in := 5, out1 => #TI_RowNr)
   END_RUNG
   RUNG wire#powerrail
      { S7_Templates := "SrcType := UInt" } EQ_Contact(in1 := "STATUS_1R5".RO01.Specific.JobNr, in2 := #CI_JobTake170Pos3)
   END_RUNG wire#w3
   RUNG wire#powerrail
      { S7_Templates := "SrcType := UInt" } EQ_Contact(in1 := "STATUS_1R5".RO01.Specific.JobNr, in2 := #CI_JobTake150Pos4)
      wire#w4
      Move(in := 7, out1 => #TI_RowNr)
   END_RUNG
   RUNG wire#powerrail
      { S7_Templates := "SrcType := UInt" } EQ_Contact(in1 := "STATUS_1R5".RO01.Specific.JobNr, in2 := #CI_JobTake170Pos4)
   END_RUNG wire#w4
   RUNG wire#powerrail
      { S7_Templates := "SrcType := UInt" } EQ_Contact(in1 := "STATUS_1R5".RO01.Specific.JobNr, in2 := #CI_JobTake150Pos5)
      wire#w5
      Move(in := 9, out1 => #TI_RowNr)
   END_RUNG
   RUNG wire#powerrail
      { S7_Templates := "SrcType := UInt" } EQ_Contact(in1 := "STATUS_1R5".RO01.Specific.JobNr, in2 := #CI_JobTake170Pos5)
   END_RUNG wire#w5
   RUNG wire#powerrail
      { S7_Templates := "SrcType := UInt" } EQ_Contact(in1 := "STATUS_1R5".RO01.Specific.JobNr, in2 := #CI_JobTake150Pos6)
      wire#w6
      Move(in := 11, out1 => #TI_RowNr)
   END_RUNG
   RUNG wire#powerrail
      { S7_Templates := "SrcType := UInt" } EQ_Contact(in1 := "STATUS_1R5".RO01.Specific.JobNr, in2 := #CI_JobTake170Pos6)
   END_RUNG wire#w6
   RUNG wire#powerrail
      { S7_Templates := "SrcType := UInt" } EQ_Contact(in1 := "STATUS_1R5".RO01.Specific.JobNr, in2 := #CI_JobTake150Pos7)
      wire#w7
      Move(in := 13, out1 => #TI_RowNr)
   END_RUNG
   RUNG wire#powerrail
      { S7_Templates := "SrcType := UInt" } EQ_Contact(in1 := "STATUS_1R5".RO01.Specific.JobNr, in2 := #CI_JobTake170Pos7)
   END_RUNG wire#w7
   RUNG wire#powerrail
      { S7_Templates := "SrcType := UInt" } EQ_Contact(in1 := "STATUS_1R5".RO01.Specific.JobNr, in2 := #CI_JobTake150Pos8)
      wire#w8
      Move(in := 15, out1 => #TI_RowNr)
   END_RUNG
   RUNG wire#powerrail
      { S7_Templates := "SrcType := UInt" } EQ_Contact(in1 := "STATUS_1R5".RO01.Specific.JobNr, in2 := #CI_JobTake170Pos8)
   END_RUNG wire#w8
   RUNG wire#powerrail
      { S7_Templates := "SrcType := UInt" } EQ_Contact(in1 := "STATUS_1R5".RO01.Specific.JobNr, in2 := #CI_JobTake150Pos9)
      wire#w9
      Move(in := 17, out1 => #TI_RowNr)
   END_RUNG
   RUNG wire#powerrail
      { S7_Templates := "SrcType := UInt" } EQ_Contact(in1 := "STATUS_1R5".RO01.Specific.JobNr, in2 := #CI_JobTake170Pos9)
   END_RUNG wire#w9
   RUNG wire#powerrail
      { S7_Templates := "SrcType := UInt" } EQ_Contact(in1 := "STATUS_1R5".RO01.Specific.JobNr, in2 := #CI_JobTake150Pos10)
      wire#w10
      Move(in := 19, out1 => #TI_RowNr)
   END_RUNG
   RUNG wire#powerrail
      { S7_Templates := "SrcType := UInt" } EQ_Contact(in1 := "STATUS_1R5".RO01.Specific.JobNr, in2 := #CI_JobTake170Pos10)
   END_RUNG wire#w10
   RUNG wire#powerrail
      { S7_Templates := "SrcType := UInt" } EQ_Contact(in1 := "STATUS_1R5".RO01.Specific.JobNr, in2 := #CI_JobTake150Pos11)
      wire#w11
      Move(in := 21, out1 => #TI_RowNr)
   END_RUNG
   RUNG wire#powerrail
      { S7_Templates := "SrcType := UInt" } EQ_Contact(in1 := "STATUS_1R5".RO01.Specific.JobNr, in2 := #CI_JobTake170Pos11)
   END_RUNG wire#w11
   RUNG wire#powerrail
      { S7_Templates := "SrcType := UInt" } EQ_Contact(in1 := "STATUS_1R5".RO01.Specific.JobNr, in2 := #CI_JobTake150Pos12)
      wire#w12
      Move(in := 23, out1 => #TI_RowNr)
   END_RUNG
   RUNG wire#powerrail
      { S7_Templates := "SrcType := UInt" } EQ_Contact(in1 := "STATUS_1R5".RO01.Specific.JobNr, in2 := #CI_JobTake170Pos12)
   END_RUNG wire#w12
   // the same network as SCL:
   IF ("STATUS_1R5".RO01.Specific.JobNr = #CI_JobTake150Pos1) OR ("STATUS_1R5".RO01.Specific.JobNr = #CI_JobTake170Pos1) THEN
       #TI_RowNr := 1;
   END_IF;
   IF ("STATUS_1R5".RO01.Specific.JobNr = #CI_JobTake150Pos2) OR ("STATUS_1R5".RO01.Specific.JobNr = #CI_JobTake170Pos2) THEN
       #TI_RowNr := 3;
   END_IF;
   IF ("STATUS_1R5".RO01.Specific.JobNr = #CI_JobTake150Pos3) OR ("STATUS_1R5".RO01.Specific.JobNr = #CI_JobTake170Pos3) THEN
       #TI_RowNr := 5;
   END_IF;
   IF ("STATUS_1R5".RO01.Specific.JobNr = #CI_JobTake150Pos4) OR ("STATUS_1R5".RO01.Specific.JobNr = #CI_JobTake170Pos4) THEN
       #TI_RowNr := 7;
   END_IF;
   IF ("STATUS_1R5".RO01.Specific.JobNr = #CI_JobTake150Pos5) OR ("STATUS_1R5".RO01.Specific.JobNr = #CI_JobTake170Pos5) THEN
       #TI_RowNr := 9;
   END_IF;
   IF ("STATUS_1R5".RO01.Specific.JobNr = #CI_JobTake150Pos6) OR ("STATUS_1R5".RO01.Specific.JobNr = #CI_JobTake170Pos6) THEN
       #TI_RowNr := 11;
   END_IF;
   IF ("STATUS_1R5".RO01.Specific.JobNr = #CI_JobTake150Pos7) OR ("STATUS_1R5".RO01.Specific.JobNr = #CI_JobTake170Pos7) THEN
       #TI_RowNr := 13;
   END_IF;
   IF ("STATUS_1R5".RO01.Specific.JobNr = #CI_JobTake150Pos8) OR ("STATUS_1R5".RO01.Specific.JobNr = #CI_JobTake170Pos8) THEN
       #TI_RowNr := 15;
   END_IF;
   IF ("STATUS_1R5".RO01.Specific.JobNr = #CI_JobTake150Pos9) OR ("STATUS_1R5".RO01.Specific.JobNr = #CI_JobTake170Pos9) THEN
       #TI_RowNr := 17;
   END_IF;
   IF ("STATUS_1R5".RO01.Specific.JobNr = #CI_JobTake150Pos10) OR ("STATUS_1R5".RO01.Specific.JobNr = #CI_JobTake170Pos10) THEN
       #TI_RowNr := 19;
   END_IF;
   IF ("STATUS_1R5".RO01.Specific.JobNr = #CI_JobTake150Pos11) OR ("STATUS_1R5".RO01.Specific.JobNr = #CI_JobTake170Pos11) THEN
       #TI_RowNr := 21;
   END_IF;
   IF ("STATUS_1R5".RO01.Specific.JobNr = #CI_JobTake150Pos12) OR ("STATUS_1R5".RO01.Specific.JobNr = #CI_JobTake170Pos12) THEN
       #TI_RowNr := 23;
   END_IF;
END_REGION

REGION Network 48: Data transfer: 150 -> 1R5
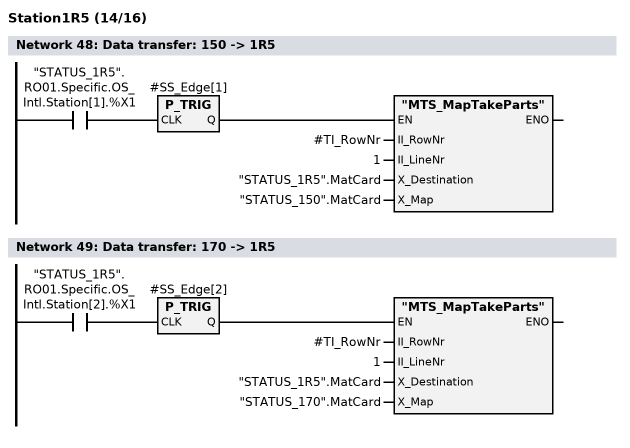
   RUNG wire#powerrail
      Contact( "STATUS_1R5".RO01.Specific.OS_Intl.Station[1].%X1 )
      P_Trig( #SS_Edge[1] )
      "MTS_MapTakeParts"(II_RowNr := #TI_RowNr, II_LineNr := 1, X_Destination := "STATUS_1R5".MatCard, X_Map := "STATUS_150".MatCard)
   END_RUNG
   // the same network as SCL:
   #_w1 := "STATUS_1R5".RO01.Specific.OS_Intl.Station[1].%X1 AND NOT #SS_Edge[1];   // rising edge
   #SS_Edge[1] := "STATUS_1R5".RO01.Specific.OS_Intl.Station[1].%X1;
   IF #_w1 THEN
       "MTS_MapTakeParts"(II_RowNr := #TI_RowNr,
                          II_LineNr := 1,
                          X_Destination := "STATUS_1R5".MatCard,
                          X_Map := "STATUS_150".MatCard);
   END_IF;
END_REGION

REGION Network 49: Data transfer: 170 -> 1R5
   RUNG wire#powerrail
      Contact( "STATUS_1R5".RO01.Specific.OS_Intl.Station[2].%X1 )
      P_Trig( #SS_Edge[2] )
      "MTS_MapTakeParts"(II_RowNr := #TI_RowNr, II_LineNr := 1, X_Destination := "STATUS_1R5".MatCard, X_Map := "STATUS_170".MatCard)
   END_RUNG
   // the same network as SCL:
   #_w1 := "STATUS_1R5".RO01.Specific.OS_Intl.Station[2].%X1 AND NOT #SS_Edge[2];   // rising edge
   #SS_Edge[2] := "STATUS_1R5".RO01.Specific.OS_Intl.Station[2].%X1;
   IF #_w1 THEN
       "MTS_MapTakeParts"(II_RowNr := #TI_RowNr,
                          II_LineNr := 1,
                          X_Destination := "STATUS_1R5".MatCard,
                          X_Map := "STATUS_170".MatCard);
   END_IF;
END_REGION

REGION Network 50: Data transfer: BSN1 - row/line number
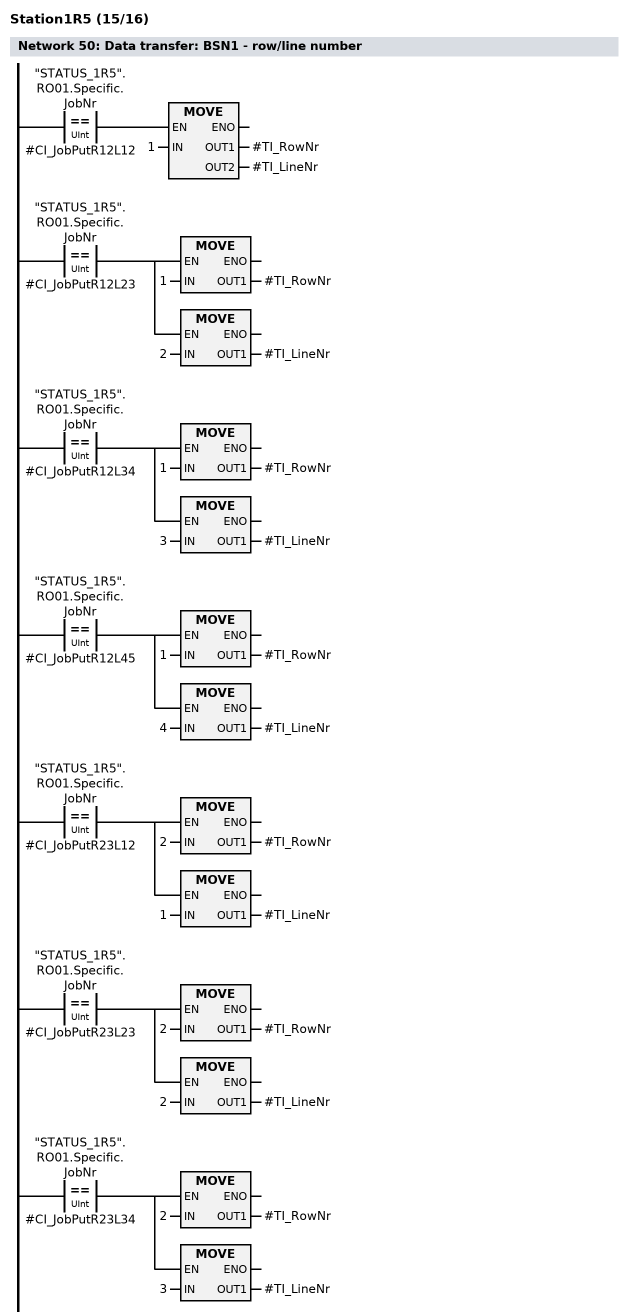
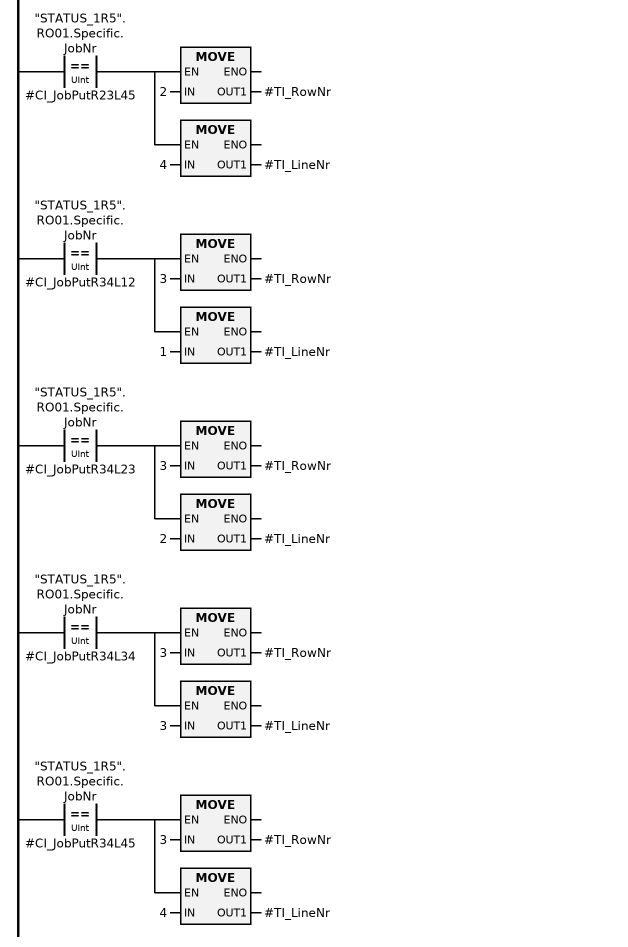
   RUNG wire#powerrail
      { S7_Templates := "SrcType := UInt" } EQ_Contact(in1 := "STATUS_1R5".RO01.Specific.JobNr, in2 := #CI_JobPutR12L12)
      Move(in := 1, out1 => #TI_RowNr, out2 => #TI_LineNr)
   END_RUNG
   RUNG wire#powerrail
      { S7_Templates := "SrcType := UInt" } EQ_Contact(in1 := "STATUS_1R5".RO01.Specific.JobNr, in2 := #CI_JobPutR12L23)
      wire#w1
      Move(in := 1, out1 => #TI_RowNr)
   END_RUNG
   RUNG wire#w1
      Move(in := 2, out1 => #TI_LineNr)
   END_RUNG
   RUNG wire#powerrail
      { S7_Templates := "SrcType := UInt" } EQ_Contact(in1 := "STATUS_1R5".RO01.Specific.JobNr, in2 := #CI_JobPutR12L34)
      wire#w2
      Move(in := 1, out1 => #TI_RowNr)
   END_RUNG
   RUNG wire#w2
      Move(in := 3, out1 => #TI_LineNr)
   END_RUNG
   RUNG wire#powerrail
      { S7_Templates := "SrcType := UInt" } EQ_Contact(in1 := "STATUS_1R5".RO01.Specific.JobNr, in2 := #CI_JobPutR12L45)
      wire#w3
      Move(in := 1, out1 => #TI_RowNr)
   END_RUNG
   RUNG wire#w3
      Move(in := 4, out1 => #TI_LineNr)
   END_RUNG
   RUNG wire#powerrail
      { S7_Templates := "SrcType := UInt" } EQ_Contact(in1 := "STATUS_1R5".RO01.Specific.JobNr, in2 := #CI_JobPutR23L12)
      wire#w4
      Move(in := 2, out1 => #TI_RowNr)
   END_RUNG
   RUNG wire#w4
      Move(in := 1, out1 => #TI_LineNr)
   END_RUNG
   RUNG wire#powerrail
      { S7_Templates := "SrcType := UInt" } EQ_Contact(in1 := "STATUS_1R5".RO01.Specific.JobNr, in2 := #CI_JobPutR23L23)
      wire#w5
      Move(in := 2, out1 => #TI_RowNr)
   END_RUNG
   RUNG wire#w5
      Move(in := 2, out1 => #TI_LineNr)
   END_RUNG
   RUNG wire#powerrail
      { S7_Templates := "SrcType := UInt" } EQ_Contact(in1 := "STATUS_1R5".RO01.Specific.JobNr, in2 := #CI_JobPutR23L34)
      wire#w6
      Move(in := 2, out1 => #TI_RowNr)
   END_RUNG
   RUNG wire#w6
      Move(in := 3, out1 => #TI_LineNr)
   END_RUNG
   RUNG wire#powerrail
      { S7_Templates := "SrcType := UInt" } EQ_Contact(in1 := "STATUS_1R5".RO01.Specific.JobNr, in2 := #CI_JobPutR23L45)
      wire#w7
      Move(in := 2, out1 => #TI_RowNr)
   END_RUNG
   RUNG wire#w7
      Move(in := 4, out1 => #TI_LineNr)
   END_RUNG
   RUNG wire#powerrail
      { S7_Templates := "SrcType := UInt" } EQ_Contact(in1 := "STATUS_1R5".RO01.Specific.JobNr, in2 := #CI_JobPutR34L12)
      wire#w8
      Move(in := 3, out1 => #TI_RowNr)
   END_RUNG
   RUNG wire#w8
      Move(in := 1, out1 => #TI_LineNr)
   END_RUNG
   RUNG wire#powerrail
      { S7_Templates := "SrcType := UInt" } EQ_Contact(in1 := "STATUS_1R5".RO01.Specific.JobNr, in2 := #CI_JobPutR34L23)
      wire#w9
      Move(in := 3, out1 => #TI_RowNr)
   END_RUNG
   RUNG wire#w9
      Move(in := 2, out1 => #TI_LineNr)
   END_RUNG
   RUNG wire#powerrail
      { S7_Templates := "SrcType := UInt" } EQ_Contact(in1 := "STATUS_1R5".RO01.Specific.JobNr, in2 := #CI_JobPutR34L34)
      wire#w10
      Move(in := 3, out1 => #TI_RowNr)
   END_RUNG
   RUNG wire#w10
      Move(in := 3, out1 => #TI_LineNr)
   END_RUNG
   RUNG wire#powerrail
      { S7_Templates := "SrcType := UInt" } EQ_Contact(in1 := "STATUS_1R5".RO01.Specific.JobNr, in2 := #CI_JobPutR34L45)
      wire#w11
      Move(in := 3, out1 => #TI_RowNr)
   END_RUNG
   RUNG wire#w11
      Move(in := 4, out1 => #TI_LineNr)
   END_RUNG
   // the same network as SCL:
   IF "STATUS_1R5".RO01.Specific.JobNr = #CI_JobPutR12L12 THEN
       #TI_RowNr := 1;
       #TI_LineNr := 1;
   END_IF;
   IF "STATUS_1R5".RO01.Specific.JobNr = #CI_JobPutR12L23 THEN
       #TI_RowNr := 1;
       #TI_LineNr := 2;
   END_IF;
   IF "STATUS_1R5".RO01.Specific.JobNr = #CI_JobPutR12L34 THEN
       #TI_RowNr := 1;
       #TI_LineNr := 3;
   END_IF;
   IF "STATUS_1R5".RO01.Specific.JobNr = #CI_JobPutR12L45 THEN
       #TI_RowNr := 1;
       #TI_LineNr := 4;
   END_IF;
   IF "STATUS_1R5".RO01.Specific.JobNr = #CI_JobPutR23L12 THEN
       #TI_RowNr := 2;
       #TI_LineNr := 1;
   END_IF;
   IF "STATUS_1R5".RO01.Specific.JobNr = #CI_JobPutR23L23 THEN
       #TI_RowNr := 2;
       #TI_LineNr := 2;
   END_IF;
   IF "STATUS_1R5".RO01.Specific.JobNr = #CI_JobPutR23L34 THEN
       #TI_RowNr := 2;
       #TI_LineNr := 3;
   END_IF;
   IF "STATUS_1R5".RO01.Specific.JobNr = #CI_JobPutR23L45 THEN
       #TI_RowNr := 2;
       #TI_LineNr := 4;
   END_IF;
   IF "STATUS_1R5".RO01.Specific.JobNr = #CI_JobPutR34L12 THEN
       #TI_RowNr := 3;
       #TI_LineNr := 1;
   END_IF;
   IF "STATUS_1R5".RO01.Specific.JobNr = #CI_JobPutR34L23 THEN
       #TI_RowNr := 3;
       #TI_LineNr := 2;
   END_IF;
   IF "STATUS_1R5".RO01.Specific.JobNr = #CI_JobPutR34L34 THEN
       #TI_RowNr := 3;
       #TI_LineNr := 3;
   END_IF;
   IF "STATUS_1R5".RO01.Specific.JobNr = #CI_JobPutR34L45 THEN
       #TI_RowNr := 3;
       #TI_LineNr := 4;
   END_IF;
END_REGION

REGION Network 51: Data transfer: 1R5 -> BSN1
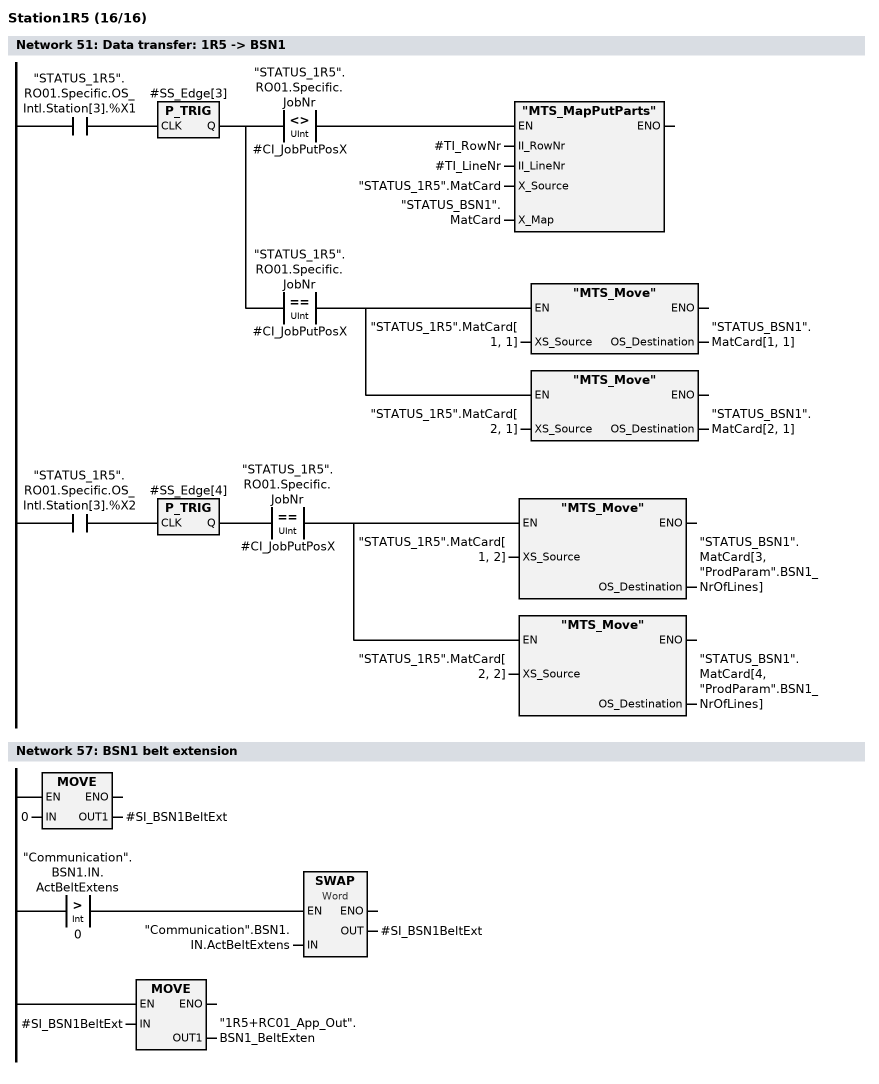
   RUNG wire#powerrail
      Contact( "STATUS_1R5".RO01.Specific.OS_Intl.Station[3].%X1 )
      P_Trig( #SS_Edge[3] )
      wire#w1
      { S7_Templates := "SrcType := UInt" } NE_Contact(in1 := "STATUS_1R5".RO01.Specific.JobNr, in2 := #CI_JobPutPosX)
      "MTS_MapPutParts"(II_RowNr := #TI_RowNr, II_LineNr := #TI_LineNr, X_Source := "STATUS_1R5".MatCard, X_Map := "STATUS_BSN1".MatCard)
   END_RUNG
   RUNG wire#w1
      { S7_Templates := "SrcType := UInt" } EQ_Contact(in1 := "STATUS_1R5".RO01.Specific.JobNr, in2 := #CI_JobPutPosX)
      wire#w2
      "MTS_Move"(XS_Source := "STATUS_1R5".MatCard[1, 1], OS_Destination => "STATUS_BSN1".MatCard[1, 1])
   END_RUNG
   RUNG wire#w2
      "MTS_Move"(XS_Source := "STATUS_1R5".MatCard[2, 1], OS_Destination => "STATUS_BSN1".MatCard[2, 1])
   END_RUNG
   RUNG wire#powerrail
      Contact( "STATUS_1R5".RO01.Specific.OS_Intl.Station[3].%X2 )
      P_Trig( #SS_Edge[4] )
      { S7_Templates := "SrcType := UInt" } EQ_Contact(in1 := "STATUS_1R5".RO01.Specific.JobNr, in2 := #CI_JobPutPosX)
      wire#w3
      "MTS_Move"(XS_Source := "STATUS_1R5".MatCard[1, 2], OS_Destination => "STATUS_BSN1".MatCard[3, "ProdParam".BSN1_NrOfLines])
   END_RUNG
   RUNG wire#w3
      "MTS_Move"(XS_Source := "STATUS_1R5".MatCard[2, 2], OS_Destination => "STATUS_BSN1".MatCard[4, "ProdParam".BSN1_NrOfLines])
   END_RUNG
   // the same network as SCL:
   #_w1 := "STATUS_1R5".RO01.Specific.OS_Intl.Station[3].%X1 AND NOT #SS_Edge[3];   // rising edge
   #SS_Edge[3] := "STATUS_1R5".RO01.Specific.OS_Intl.Station[3].%X1;
   IF #_w1 AND ("STATUS_1R5".RO01.Specific.JobNr <> #CI_JobPutPosX) THEN
       "MTS_MapPutParts"(II_RowNr := #TI_RowNr,
                         II_LineNr := #TI_LineNr,
                         X_Source := "STATUS_1R5".MatCard,
                         X_Map := "STATUS_BSN1".MatCard);
   END_IF;
   #_w2 := #_w1 AND ("STATUS_1R5".RO01.Specific.JobNr = #CI_JobPutPosX);
   IF #_w2 THEN
       "MTS_Move"(XS_Source := "STATUS_1R5".MatCard[1, 1], OS_Destination => "STATUS_BSN1".MatCard[1, 1]);
       "MTS_Move"(XS_Source := "STATUS_1R5".MatCard[2, 1], OS_Destination => "STATUS_BSN1".MatCard[2, 1]);
   END_IF;
   #_w3 := "STATUS_1R5".RO01.Specific.OS_Intl.Station[3].%X2 AND NOT #SS_Edge[4];   // rising edge
   #SS_Edge[4] := "STATUS_1R5".RO01.Specific.OS_Intl.Station[3].%X2;
   #_w4 := #_w3 AND ("STATUS_1R5".RO01.Specific.JobNr = #CI_JobPutPosX);
   IF #_w4 THEN
       "MTS_Move"(XS_Source := "STATUS_1R5".MatCard[1, 2],
                  OS_Destination => "STATUS_BSN1".MatCard[3, "ProdParam".BSN1_NrOfLines]);
       "MTS_Move"(XS_Source := "STATUS_1R5".MatCard[2, 2],
                  OS_Destination => "STATUS_BSN1".MatCard[4, "ProdParam".BSN1_NrOfLines]);
   END_IF;
END_REGION

REGION Network 52: *************** Aplication Interface ***************
END_REGION

REGION Network 53 (SCL): Prediction part on position 1
   "1R5+RC01_App_Out"."150/170 - part in position 1" :=
   ("STATUS_1R5".RO01.Specific.JobNr = #CI_JobTake150Pos1) AND "STATUS_150".MatCard[1, 1].Occupied
   OR ("STATUS_1R5".RO01.Specific.JobNr = #CI_JobTake150Pos2) AND "STATUS_150".MatCard[3, 1].Occupied
   OR ("STATUS_1R5".RO01.Specific.JobNr = #CI_JobTake150Pos3) AND "STATUS_150".MatCard[5, 1].Occupied
   OR ("STATUS_1R5".RO01.Specific.JobNr = #CI_JobTake150Pos4) AND "STATUS_150".MatCard[7, 1].Occupied
   OR ("STATUS_1R5".RO01.Specific.JobNr = #CI_JobTake150Pos5) AND "STATUS_150".MatCard[9, 1].Occupied
   OR ("STATUS_1R5".RO01.Specific.JobNr = #CI_JobTake150Pos6) AND "STATUS_150".MatCard[11, 1].Occupied
   OR ("STATUS_1R5".RO01.Specific.JobNr = #CI_JobTake150Pos7) AND "STATUS_150".MatCard[13, 1].Occupied
   OR ("STATUS_1R5".RO01.Specific.JobNr = #CI_JobTake150Pos8) AND "STATUS_150".MatCard[15, 1].Occupied
   OR ("STATUS_1R5".RO01.Specific.JobNr = #CI_JobTake150Pos9) AND "STATUS_150".MatCard[17, 1].Occupied
   OR ("STATUS_1R5".RO01.Specific.JobNr = #CI_JobTake150Pos10) AND "STATUS_150".MatCard[19, 1].Occupied
   OR ("STATUS_1R5".RO01.Specific.JobNr = #CI_JobTake150Pos11) AND "STATUS_150".MatCard[21, 1].Occupied
   OR ("STATUS_1R5".RO01.Specific.JobNr = #CI_JobTake150Pos12) AND "STATUS_150".MatCard[23, 1].Occupied
   OR ("STATUS_1R5".RO01.Specific.JobNr = #CI_JobTake170Pos1) AND "STATUS_170".MatCard[1, 1].Occupied
   OR ("STATUS_1R5".RO01.Specific.JobNr = #CI_JobTake170Pos2) AND "STATUS_170".MatCard[3, 1].Occupied
   OR ("STATUS_1R5".RO01.Specific.JobNr = #CI_JobTake170Pos3) AND "STATUS_170".MatCard[5, 1].Occupied
   OR ("STATUS_1R5".RO01.Specific.JobNr = #CI_JobTake170Pos4) AND "STATUS_170".MatCard[7, 1].Occupied
   OR ("STATUS_1R5".RO01.Specific.JobNr = #CI_JobTake170Pos5) AND "STATUS_170".MatCard[9, 1].Occupied
   OR ("STATUS_1R5".RO01.Specific.JobNr = #CI_JobTake170Pos6) AND "STATUS_170".MatCard[11, 1].Occupied
   OR ("STATUS_1R5".RO01.Specific.JobNr = #CI_JobTake170Pos7) AND "STATUS_170".MatCard[13, 1].Occupied
   OR ("STATUS_1R5".RO01.Specific.JobNr = #CI_JobTake170Pos8) AND "STATUS_170".MatCard[15, 1].Occupied
   OR ("STATUS_1R5".RO01.Specific.JobNr = #CI_JobTake170Pos9) AND "STATUS_170".MatCard[17, 1].Occupied
   OR ("STATUS_1R5".RO01.Specific.JobNr = #CI_JobTake170Pos10) AND "STATUS_170".MatCard[19, 1].Occupied
   OR ("STATUS_1R5".RO01.Specific.JobNr = #CI_JobTake170Pos11) AND "STATUS_170".MatCard[21, 1].Occupied
   OR ("STATUS_1R5".RO01.Specific.JobNr = #CI_JobTake170Pos12) AND "STATUS_170".MatCard[23, 1].Occupied;
END_REGION

REGION Network 54 (SCL): Prediction part on position 2
   "1R5+RC01_App_Out"."150/170 - part in position 2" :=
   ("STATUS_1R5".RO01.Specific.JobNr = #CI_JobTake150Pos1) AND "STATUS_150".MatCard[1, 2].Occupied
   OR ("STATUS_1R5".RO01.Specific.JobNr = #CI_JobTake150Pos2) AND "STATUS_150".MatCard[3, 2].Occupied
   OR ("STATUS_1R5".RO01.Specific.JobNr = #CI_JobTake150Pos3) AND "STATUS_150".MatCard[5, 2].Occupied
   OR ("STATUS_1R5".RO01.Specific.JobNr = #CI_JobTake150Pos4) AND "STATUS_150".MatCard[7, 2].Occupied
   OR ("STATUS_1R5".RO01.Specific.JobNr = #CI_JobTake150Pos5) AND "STATUS_150".MatCard[9, 2].Occupied
   OR ("STATUS_1R5".RO01.Specific.JobNr = #CI_JobTake150Pos6) AND "STATUS_150".MatCard[11, 2].Occupied
   OR ("STATUS_1R5".RO01.Specific.JobNr = #CI_JobTake150Pos7) AND "STATUS_150".MatCard[13, 2].Occupied
   OR ("STATUS_1R5".RO01.Specific.JobNr = #CI_JobTake150Pos8) AND "STATUS_150".MatCard[15, 2].Occupied
   OR ("STATUS_1R5".RO01.Specific.JobNr = #CI_JobTake150Pos9) AND "STATUS_150".MatCard[17, 2].Occupied
   OR ("STATUS_1R5".RO01.Specific.JobNr = #CI_JobTake150Pos10) AND "STATUS_150".MatCard[19, 2].Occupied
   OR ("STATUS_1R5".RO01.Specific.JobNr = #CI_JobTake150Pos11) AND "STATUS_150".MatCard[21, 2].Occupied
   OR ("STATUS_1R5".RO01.Specific.JobNr = #CI_JobTake150Pos12) AND "STATUS_150".MatCard[23, 2].Occupied
   OR ("STATUS_1R5".RO01.Specific.JobNr = #CI_JobTake170Pos1) AND "STATUS_170".MatCard[1, 2].Occupied
   OR ("STATUS_1R5".RO01.Specific.JobNr = #CI_JobTake170Pos2) AND "STATUS_170".MatCard[3, 2].Occupied
   OR ("STATUS_1R5".RO01.Specific.JobNr = #CI_JobTake170Pos3) AND "STATUS_170".MatCard[5, 2].Occupied
   OR ("STATUS_1R5".RO01.Specific.JobNr = #CI_JobTake170Pos4) AND "STATUS_170".MatCard[7, 2].Occupied
   OR ("STATUS_1R5".RO01.Specific.JobNr = #CI_JobTake170Pos5) AND "STATUS_170".MatCard[9, 2].Occupied
   OR ("STATUS_1R5".RO01.Specific.JobNr = #CI_JobTake170Pos6) AND "STATUS_170".MatCard[11, 2].Occupied
   OR ("STATUS_1R5".RO01.Specific.JobNr = #CI_JobTake170Pos7) AND "STATUS_170".MatCard[13, 2].Occupied
   OR ("STATUS_1R5".RO01.Specific.JobNr = #CI_JobTake170Pos8) AND "STATUS_170".MatCard[15, 2].Occupied
   OR ("STATUS_1R5".RO01.Specific.JobNr = #CI_JobTake170Pos9) AND "STATUS_170".MatCard[17, 2].Occupied
   OR ("STATUS_1R5".RO01.Specific.JobNr = #CI_JobTake170Pos10) AND "STATUS_170".MatCard[19, 2].Occupied
   OR ("STATUS_1R5".RO01.Specific.JobNr = #CI_JobTake170Pos11) AND "STATUS_170".MatCard[21, 2].Occupied
   OR ("STATUS_1R5".RO01.Specific.JobNr = #CI_JobTake170Pos12) AND "STATUS_170".MatCard[23, 2].Occupied;
END_REGION

REGION Network 55 (SCL): Prediction part on position 3
   "1R5+RC01_App_Out"."150/170 - part in position 3" :=
   ("STATUS_1R5".RO01.Specific.JobNr = #CI_JobTake150Pos1) AND "STATUS_150".MatCard[2, 1].Occupied
   OR ("STATUS_1R5".RO01.Specific.JobNr = #CI_JobTake150Pos2) AND "STATUS_150".MatCard[4, 1].Occupied
   OR ("STATUS_1R5".RO01.Specific.JobNr = #CI_JobTake150Pos3) AND "STATUS_150".MatCard[6, 1].Occupied
   OR ("STATUS_1R5".RO01.Specific.JobNr = #CI_JobTake150Pos4) AND "STATUS_150".MatCard[8, 1].Occupied
   OR ("STATUS_1R5".RO01.Specific.JobNr = #CI_JobTake150Pos5) AND "STATUS_150".MatCard[10, 1].Occupied
   OR ("STATUS_1R5".RO01.Specific.JobNr = #CI_JobTake150Pos6) AND "STATUS_150".MatCard[12, 1].Occupied
   OR ("STATUS_1R5".RO01.Specific.JobNr = #CI_JobTake150Pos7) AND "STATUS_150".MatCard[14, 1].Occupied
   OR ("STATUS_1R5".RO01.Specific.JobNr = #CI_JobTake150Pos8) AND "STATUS_150".MatCard[16, 1].Occupied
   OR ("STATUS_1R5".RO01.Specific.JobNr = #CI_JobTake150Pos9) AND "STATUS_150".MatCard[18, 1].Occupied
   OR ("STATUS_1R5".RO01.Specific.JobNr = #CI_JobTake150Pos10) AND "STATUS_150".MatCard[20, 1].Occupied
   OR ("STATUS_1R5".RO01.Specific.JobNr = #CI_JobTake150Pos11) AND "STATUS_150".MatCard[22, 1].Occupied
   OR ("STATUS_1R5".RO01.Specific.JobNr = #CI_JobTake150Pos12) AND "STATUS_150".MatCard[24, 1].Occupied
   OR ("STATUS_1R5".RO01.Specific.JobNr = #CI_JobTake170Pos1) AND "STATUS_170".MatCard[2, 1].Occupied
   OR ("STATUS_1R5".RO01.Specific.JobNr = #CI_JobTake170Pos2) AND "STATUS_170".MatCard[4, 1].Occupied
   OR ("STATUS_1R5".RO01.Specific.JobNr = #CI_JobTake170Pos3) AND "STATUS_170".MatCard[6, 1].Occupied
   OR ("STATUS_1R5".RO01.Specific.JobNr = #CI_JobTake170Pos4) AND "STATUS_170".MatCard[8, 1].Occupied
   OR ("STATUS_1R5".RO01.Specific.JobNr = #CI_JobTake170Pos5) AND "STATUS_170".MatCard[10, 1].Occupied
   OR ("STATUS_1R5".RO01.Specific.JobNr = #CI_JobTake170Pos6) AND "STATUS_170".MatCard[12, 1].Occupied
   OR ("STATUS_1R5".RO01.Specific.JobNr = #CI_JobTake170Pos7) AND "STATUS_170".MatCard[14, 1].Occupied
   OR ("STATUS_1R5".RO01.Specific.JobNr = #CI_JobTake170Pos8) AND "STATUS_170".MatCard[16, 1].Occupied
   OR ("STATUS_1R5".RO01.Specific.JobNr = #CI_JobTake170Pos9) AND "STATUS_170".MatCard[18, 1].Occupied
   OR ("STATUS_1R5".RO01.Specific.JobNr = #CI_JobTake170Pos10) AND "STATUS_170".MatCard[20, 1].Occupied
   OR ("STATUS_1R5".RO01.Specific.JobNr = #CI_JobTake170Pos11) AND "STATUS_170".MatCard[22, 1].Occupied
   OR ("STATUS_1R5".RO01.Specific.JobNr = #CI_JobTake170Pos12) AND "STATUS_170".MatCard[24, 1].Occupied;
END_REGION

REGION Network 56 (SCL): Prediction part on position 4
   "1R5+RC01_App_Out"."150/170 - part in position 4" :=
   ("STATUS_1R5".RO01.Specific.JobNr = #CI_JobTake150Pos1) AND "STATUS_150".MatCard[2, 2].Occupied
   OR ("STATUS_1R5".RO01.Specific.JobNr = #CI_JobTake150Pos2) AND "STATUS_150".MatCard[4, 2].Occupied
   OR ("STATUS_1R5".RO01.Specific.JobNr = #CI_JobTake150Pos3) AND "STATUS_150".MatCard[6, 2].Occupied
   OR ("STATUS_1R5".RO01.Specific.JobNr = #CI_JobTake150Pos4) AND "STATUS_150".MatCard[8, 2].Occupied
   OR ("STATUS_1R5".RO01.Specific.JobNr = #CI_JobTake150Pos5) AND "STATUS_150".MatCard[10, 2].Occupied
   OR ("STATUS_1R5".RO01.Specific.JobNr = #CI_JobTake150Pos6) AND "STATUS_150".MatCard[12, 2].Occupied
   OR ("STATUS_1R5".RO01.Specific.JobNr = #CI_JobTake150Pos7) AND "STATUS_150".MatCard[14, 2].Occupied
   OR ("STATUS_1R5".RO01.Specific.JobNr = #CI_JobTake150Pos8) AND "STATUS_150".MatCard[16, 2].Occupied
   OR ("STATUS_1R5".RO01.Specific.JobNr = #CI_JobTake150Pos9) AND "STATUS_150".MatCard[18, 2].Occupied
   OR ("STATUS_1R5".RO01.Specific.JobNr = #CI_JobTake150Pos10) AND "STATUS_150".MatCard[20, 2].Occupied
   OR ("STATUS_1R5".RO01.Specific.JobNr = #CI_JobTake150Pos11) AND "STATUS_150".MatCard[22, 2].Occupied
   OR ("STATUS_1R5".RO01.Specific.JobNr = #CI_JobTake150Pos12) AND "STATUS_150".MatCard[24, 2].Occupied
   OR ("STATUS_1R5".RO01.Specific.JobNr = #CI_JobTake170Pos1) AND "STATUS_170".MatCard[2, 2].Occupied
   OR ("STATUS_1R5".RO01.Specific.JobNr = #CI_JobTake170Pos2) AND "STATUS_170".MatCard[4, 2].Occupied
   OR ("STATUS_1R5".RO01.Specific.JobNr = #CI_JobTake170Pos3) AND "STATUS_170".MatCard[6, 2].Occupied
   OR ("STATUS_1R5".RO01.Specific.JobNr = #CI_JobTake170Pos4) AND "STATUS_170".MatCard[8, 2].Occupied
   OR ("STATUS_1R5".RO01.Specific.JobNr = #CI_JobTake170Pos5) AND "STATUS_170".MatCard[10, 2].Occupied
   OR ("STATUS_1R5".RO01.Specific.JobNr = #CI_JobTake170Pos6) AND "STATUS_170".MatCard[12, 2].Occupied
   OR ("STATUS_1R5".RO01.Specific.JobNr = #CI_JobTake170Pos7) AND "STATUS_170".MatCard[14, 2].Occupied
   OR ("STATUS_1R5".RO01.Specific.JobNr = #CI_JobTake170Pos8) AND "STATUS_170".MatCard[16, 2].Occupied
   OR ("STATUS_1R5".RO01.Specific.JobNr = #CI_JobTake170Pos9) AND "STATUS_170".MatCard[18, 2].Occupied
   OR ("STATUS_1R5".RO01.Specific.JobNr = #CI_JobTake170Pos10) AND "STATUS_170".MatCard[20, 2].Occupied
   OR ("STATUS_1R5".RO01.Specific.JobNr = #CI_JobTake170Pos11) AND "STATUS_170".MatCard[22, 2].Occupied
   OR ("STATUS_1R5".RO01.Specific.JobNr = #CI_JobTake170Pos12) AND "STATUS_170".MatCard[24, 2].Occupied;
END_REGION

REGION Network 57: BSN1 belt extension
   #SI_BSN1BeltExt := 0;
   IF "Communication".BSN1.IN.ActBeltExtens > 0 THEN
       #SI_BSN1BeltExt := SWAP("Communication".BSN1.IN.ActBeltExtens);
   END_IF;
   "1R5+RC01_App_Out".BSN1_BeltExten := #SI_BSN1BeltExt;
END_REGION
END_FUNCTION_BLOCK
